# B&R Automation Studio project Kesim (part 4)

#### ManuelAxis.st
```iecst
(*********************************************************************************
 * Copyright:
 * Author:    baranc
 * Created:   October 16, 2025/1:34 PM
 *********************************************************************************)

ACTION ManuelAxis:

	//==================================================
	//		eksenlerin hatalarýnýn sýfýrlanmasý.
	//==================================================
	IF gCommUnit.Main.In.MachineReset THEN
		FOR _i:=0 TO MAX_AX_NR_MIN1 DO
			IF gAxBasic[_i].Error THEN
				gAxBasic[_i].ErrorReset := TRUE;
			END_IF;

		END_FOR
	ELSE
		FOR _i:=0 TO MAX_AX_NR_MIN1 DO
			IF EDGEPOS(gAxBasic[_i].Error = FALSE) THEN //mo25.11.29
				gAxBasic[_i].ErrorReset := FALSE;
			END_IF;
		END_FOR
	END_IF;

	//==================================================
	//		Speed Override
	//==================================================

	gHMI.Diagnosis.SpeedOverride := LREAL_TO_REAL( fbDepthSpeedOverride_0.Out.VelocityOverride) ;

	//==================================================
	//		Aktuel Kenar Hizi
	//==================================================

	IF(gAxBasic[AX_VACUUM].Velocity <> 0 AND gAxBasic[AX_HEAD_Y].Velocity = 0) THEN // movement just in X direction
		gHMI.Diagnosis.ActSealingSpeed := gAxBasic[AX_VACUUM].Velocity;
		IF gAxBasic[AX_VACUUM].Velocity > 1 THEN
	  		gHMI.Widget.MoveHead.Image		:= 'Media/CMS/right.png' ;
		ELSIF gAxBasic[AX_VACUUM].Velocity < -1		THEN

			gHMI.Widget.MoveHead.Image		:= 'Media/CMS/left.png' ;
		END_IF;
	ELSIF (gAxBasic[AX_HEAD_Y].Velocity <> 0 AND gAxBasic[AX_VACUUM].Velocity = 0) THEN // movement just in Y direction
		gHMI.Diagnosis.ActSealingSpeed  := gAxBasic[AX_HEAD_Y].Velocity;
		IF gAxBasic[AX_HEAD_Y].Velocity > 1 THEN
			gHMI.Widget.MoveHead.Image		:= 'Media/CMS/up.png' ;
		ELSIF gAxBasic[AX_HEAD_Y].Velocity < -1		THEN
			gHMI.Widget.MoveHead.Image		:= 'Media/CMS/down.png' ;
		END_IF;
	ELSE	// any other situation - both axes are without motion or moving together - dyn. speed is 0
		gHMI.Diagnosis.ActSealingSpeed  := 0;
		gHMI.Widget.MoveHead.Image		:= 'Media/CMS/none2.png' ;
	END_IF // end of dynamic speed

	//==================================================
	//		Manual hiz ve pos için gerekli degskenlerin atanmasi.
	//==================================================
	IF gPML[0].ModeID = PML_MODE_MAN AND gPML[0].StateCurrent = mpPACKML_STATE_IDLE  THEN

		FOR _i:=0  TO MAX_AX_NR_MIN1 DO
			IF _i >= AX_ENTRY1 AND _i <= AX_EXIT8 THEN //bc25.10.15
				IF (Loc.SelectedStatus.Entrys OR Loc.SelectedStatus.Exits) AND gHMI.Selected.Ax[AX_VACUUM] THEN // Vacuum with conveyors speed

					gAxBasicPar[_i].Velocity 	 		:= gRecData.Manual.Ax[AX_VACUUM].Speed;
					gAxBasicPar[_i].Jog.Velocity 		:= gRecData.Manual.Ax[AX_VACUUM].Speed;
					gAxBasicPar[_i].Jog.Acceleration	:= gRecData.Manual.Ax[AX_VACUUM].Speed * gACCFactor;
					gAxBasicPar[_i].Jog.Deceleration 	:= gRecData.Manual.Ax[AX_VACUUM].Speed * gACCFactor;
					gAxBasicPar[_i].Deceleration 		:= gRecData.Manual.Ax[AX_VACUUM].Speed * gACCFactor;
					gAxBasicPar[_i].Acceleration 		:= gRecData.Manual.Ax[AX_VACUUM].Speed * gACCFactor;
				ELSE
					gAxBasicPar[_i].Velocity 	 		:= gRecData.Manual.Ax[AX_ENTRY1].Speed;
					gAxBasicPar[_i].Jog.Velocity 		:= gRecData.Manual.Ax[AX_ENTRY1].Speed;
					gAxBasicPar[_i].Jog.Acceleration	:= gRecData.Manual.Ax[AX_ENTRY1].Speed * gACCFactor;
					gAxBasicPar[_i].Jog.Deceleration 	:= gRecData.Manual.Ax[AX_ENTRY1].Speed * gACCFactor;
					gAxBasicPar[_i].Deceleration 		:= gRecData.Manual.Ax[AX_ENTRY1].Speed * gACCFactor;
					gAxBasicPar[_i].Acceleration 		:= gRecData.Manual.Ax[AX_ENTRY1].Speed * gACCFactor;
				END_IF;

			ELSIF _i <> AX_HYD THEN
				IF NOT gCommUnit.Main.Status.HYD_MIXER_Y_C_AX AND ( _i = AX_HEAD_C OR _i = AX_HEAD_Y) THEN
					gAxBasicPar[_i].Velocity  			 := gRecData.Manual.Ax[_i].Speed;
					gAxBasicPar[_i].Jog.Velocity 		 := gRecData.Manual.Ax[_i].Speed;
					gAxBasicPar[_i].Jog.Acceleration 	 := gRecData.Manual.Ax[_i].Speed * gACCFactor ;
					gAxBasicPar[_i].Jog.Deceleration 	 := gRecData.Manual.Ax[_i].Speed * gACCFactor ;
					gAxBasicPar[_i].Position    		 := gRecData.Manual.Ax[_i].Pos ;
					gAxBasicPar[_i].Deceleration		 := gRecData.Manual.Ax[_i].Speed * gACCFactor ;
					gAxBasicPar[_i].Acceleration		 := gRecData.Manual.Ax[_i].Speed * gACCFactor ;
				ELSIF ( _i <> AX_HEAD_C OR _i <> AX_HEAD_Y) THEN
					gAxBasicPar[_i].Velocity  			 := gRecData.Manual.Ax[_i].Speed;
					gAxBasicPar[_i].Jog.Velocity 		 := gRecData.Manual.Ax[_i].Speed;
					gAxBasicPar[_i].Jog.Acceleration 	 := gRecData.Manual.Ax[_i].Speed * gACCFactor ;
					gAxBasicPar[_i].Jog.Deceleration 	 := gRecData.Manual.Ax[_i].Speed * gACCFactor ;
					gAxBasicPar[_i].Position    		 := gRecData.Manual.Ax[_i].Pos ;
					gAxBasicPar[_i].Deceleration		 := gRecData.Manual.Ax[_i].Speed * gACCFactor ;
					gAxBasicPar[_i].Acceleration		 := gRecData.Manual.Ax[_i].Speed * gACCFactor ;
				END_IF;

			END_IF;

		END_FOR;
		IF  gPML[0].ModeID = PML_MODE_MAN AND gPML[0].StateCurrent = mpPACKML_STATE_IDLE THEN
			IF gRecData.Manual.Ax[AX_EXIT1_BRIDGE_Y].Pos < gFixData.Ax[AX_EXIT1_BRIDGE_Y].Par.Homing.Position THEN
				gRecData.Manual.Ax[AX_EXIT1_BRIDGE_Y].Pos := LREAL_TO_REAL(gFixData.Ax[AX_EXIT1_BRIDGE_Y].Par.Homing.Position);
			END_IF;
		END_IF;

		fbExitBridgeCtrl_0[AS_BRIDGE_EXIT2].In.Parm.Position.Set 	:= gRecData.Manual.Bridge[AS_BRIDGE_EXIT2].Pos;
		fbExitBridgeCtrl_0[AS_BRIDGE_EXIT2].In.Parm.Speed.SpeedMan 	:= gRecData.Manual.Ax[AX_EXIT1_BRIDGE_Y].Speed * 0.25; // servo eksenin max hizi ile asenktron eksenin max hizi arasindaki oran

		fbExitBridgeCtrl_0[AS_BRIDGE_EXIT3].In.Parm.Position.Set 	:= gRecData.Manual.Bridge[AS_BRIDGE_EXIT3].Pos;
		fbExitBridgeCtrl_0[AS_BRIDGE_EXIT3].In.Parm.Speed.SpeedMan 	:= gRecData.Manual.Ax[AX_EXIT1_BRIDGE_Y].Speed * 0.25;

		fbExitBridgeCtrl_0[AS_BRIDGE_EXIT4].In.Parm.Position.Set 	:= gRecData.Manual.Bridge[AS_BRIDGE_EXIT4].Pos;
		fbExitBridgeCtrl_0[AS_BRIDGE_EXIT4].In.Parm.Speed.SpeedMan 	:= gRecData.Manual.Ax[AX_EXIT1_BRIDGE_Y].Speed * 0.25;

	END_IF

	//==================================================
	//		Y EKSEN GUVENLI POZISYONDA DEGIL. EXIT 1 IN YADA ENTRY 1 OUT SENSORU GORURSE VAKUM VE KONVEYOR HIZLARI DÜSSSÜN.
	//==================================================
	IF gAxBasic[AX_HEAD_Y].Position >10 AND gPML[0].ModeID = PML_MODE_MAN THEN
		IF gIO.In.Entry[ENTR1_UNIT].OutSens OR gIO.In.Exit[EXIT1_UNIT].Conv.InSens THEN
			IF gHMI.Selected.Ax[AX_VACUUM] AND gIO.In.Sealing.X2VacuumOK THEN
				gRecData.Manual.Ax[AX_VACUUM].Speed		:= 50 ;
				IF gAxBasic[AX_VACUUM].MoveActive AND gAxBasicPar[AX_VACUUM].Velocity <> gRecData.Manual.Ax[AX_VACUUM].Speed THEN

					gAxBasicPar[AX_VACUUM].Velocity 	 		:= gRecData.Manual.Ax[AX_VACUUM].Speed;
					gAxBasicPar[AX_VACUUM].Jog.Velocity 		:= gRecData.Manual.Ax[AX_VACUUM].Speed;
					gAxBasicPar[AX_VACUUM].Jog.Acceleration		:= gRecData.Manual.Ax[AX_VACUUM].Speed * 5;
					gAxBasicPar[AX_VACUUM].Jog.Deceleration 	:= gRecData.Manual.Ax[AX_VACUUM].Speed * 5;
					gAxBasicPar[AX_VACUUM].Deceleration 		:= gRecData.Manual.Ax[AX_VACUUM].Speed * 5;
					gAxBasicPar[AX_VACUUM].Acceleration 		:= gRecData.Manual.Ax[AX_VACUUM].Speed * 5;

					gAxBasicPar[AX_ENTRY1].Velocity 	 		:= gRecData.Manual.Ax[AX_VACUUM].Speed;
					gAxBasicPar[AX_ENTRY1].Jog.Velocity 		:= gRecData.Manual.Ax[AX_VACUUM].Speed;
					gAxBasicPar[AX_ENTRY1].Jog.Acceleration		:= gRecData.Manual.Ax[AX_VACUUM].Speed * 5;
					gAxBasicPar[AX_ENTRY1].Jog.Deceleration 	:= gRecData.Manual.Ax[AX_VACUUM].Speed * 5;
					gAxBasicPar[AX_ENTRY1].Deceleration 		:= gRecData.Manual.Ax[AX_VACUUM].Speed * 5;
					gAxBasicPar[AX_ENTRY1].Acceleration 		:= gRecData.Manual.Ax[AX_VACUUM].Speed * 5;

					gAxBasicPar[AX_EXIT1].Velocity 	 			:= gRecData.Manual.Ax[AX_VACUUM].Speed;
					gAxBasicPar[AX_EXIT1].Jog.Velocity 			:= gRecData.Manual.Ax[AX_VACUUM].Speed;
					gAxBasicPar[AX_EXIT1].Jog.Acceleration		:= gRecData.Manual.Ax[AX_VACUUM].Speed * 5;
					gAxBasicPar[AX_EXIT1].Jog.Deceleration 		:= gRecData.Manual.Ax[AX_VACUUM].Speed * 5;
					gAxBasicPar[AX_EXIT1].Deceleration 			:= gRecData.Manual.Ax[AX_VACUUM].Speed * 5;
					gAxBasicPar[AX_EXIT1].Acceleration 			:= gRecData.Manual.Ax[AX_VACUUM].Speed * 5;

					IF (gAxBasic[AX_VACUUM].MoveActive AND gAxBasicPar[AX_VACUUM].Velocity <> gAxBasic[AX_VACUUM].Velocity)  THEN
						gAxBasic[AX_VACUUM].Update 	:= TRUE ;
					END_IF;

					IF (gAxBasic[AX_ENTRY1].MoveActive AND gAxBasicPar[AX_ENTRY1].Velocity <> gAxBasic[AX_ENTRY1].Velocity)  THEN
						gAxBasic[AX_ENTRY1].Update 	:= TRUE ;
					END_IF;

					IF (gAxBasic[AX_EXIT1].MoveActive AND gAxBasicPar[AX_EXIT1].Velocity <> gAxBasic[AX_EXIT1].Velocity) THEN
						gAxBasic[AX_EXIT1].Update	:= TRUE ;
					END_IF;
				END_IF
				IF gAxBasic[AX_VACUUM].UpdateDone THEN
					gAxBasic[AX_VACUUM].Update 	:= FALSE ;
				END_IF;
				IF gAxBasic[AX_ENTRY1].UpdateDone THEN
					gAxBasic[AX_ENTRY1].Update 	:= FALSE ;
				END_IF;
				IF gAxBasic[AX_EXIT1].UpdateDone THEN
					gAxBasic[AX_EXIT1].Update	:= FALSE ;
				END_IF;

			ELSIF gHMI.Selected.Ax[AX_ENTRY1] OR gHMI.Selected.Ax[AX_EXIT1] THEN
				gRecData.Manual.Ax[AX_ENTRY1].Speed		:= 50 ;

				gAxBasicPar[AX_ENTRY1].Velocity 	 		:= gRecData.Manual.Ax[AX_ENTRY1].Speed;
				gAxBasicPar[AX_ENTRY1].Jog.Velocity 		:= gRecData.Manual.Ax[AX_ENTRY1].Speed;
				gAxBasicPar[AX_ENTRY1].Jog.Acceleration		:= gRecData.Manual.Ax[AX_ENTRY1].Speed * 5;
				gAxBasicPar[AX_ENTRY1].Jog.Deceleration 	:= gRecData.Manual.Ax[AX_ENTRY1].Speed * 5;
				gAxBasicPar[AX_ENTRY1].Deceleration 		:= gRecData.Manual.Ax[AX_ENTRY1].Speed * 5;
				gAxBasicPar[AX_ENTRY1].Acceleration 		:= gRecData.Manual.Ax[AX_ENTRY1].Speed * 5;

				gAxBasicPar[AX_EXIT1].Velocity 	 			:= gRecData.Manual.Ax[AX_ENTRY1].Speed;
				gAxBasicPar[AX_EXIT1].Jog.Velocity 			:= gRecData.Manual.Ax[AX_ENTRY1].Speed;
				gAxBasicPar[AX_EXIT1].Jog.Acceleration		:= gRecData.Manual.Ax[AX_ENTRY1].Speed * 5;
				gAxBasicPar[AX_EXIT1].Jog.Deceleration 		:= gRecData.Manual.Ax[AX_ENTRY1].Speed * 5;
				gAxBasicPar[AX_EXIT1].Deceleration 			:= gRecData.Manual.Ax[AX_ENTRY1].Speed * 5;
				gAxBasicPar[AX_EXIT1].Acceleration 			:= gRecData.Manual.Ax[AX_ENTRY1].Speed * 5;

				IF (gAxBasic[AX_ENTRY1].MoveActive AND gAxBasicPar[AX_ENTRY1].Velocity <> gAxBasic[AX_ENTRY1].Velocity)  THEN
					gAxBasic[AX_ENTRY1].Update 	:= TRUE ;
				END_IF;

				IF (gAxBasic[AX_EXIT1].MoveActive AND gAxBasicPar[AX_EXIT1].Velocity <> gAxBasic[AX_EXIT1].Velocity) THEN
					gAxBasic[AX_EXIT1].Update	:= TRUE ;
				END_IF;
				IF gAxBasic[AX_ENTRY1].UpdateDone THEN
					gAxBasic[AX_ENTRY1].Update 	:= FALSE ;
				END_IF;
				IF gAxBasic[AX_EXIT1].UpdateDone THEN
					gAxBasic[AX_EXIT1].Update	:= FALSE ;
				END_IF;
			END_IF;

		END_IF;
	END_IF;
	//	gAxBasicPar[AX_EXIT1]();
	//	gAxBasic[AX_EXIT1]();

	//==================================================
	//		EXIT CONV SEÇILI MI ?
	//==================================================
	Loc.SelectedStatus.Exits := FALSE;
	FOR _i := AX_EXIT1 TO AX_EXIT8 DO

		IF gHMI.Selected.Ax[_i] THEN
			Loc.SelectedStatus.Exits := TRUE;
		END_IF;

	END_FOR;

	//==================================================
	//		ENTRY CONV SEÇILI MI ?
	//==================================================
	Loc.SelectedStatus.Entrys := FALSE;
	FOR _i:=AX_ENTRY1 TO AX_ENTRY4 DO

		IF gHMI.Selected.Ax[_i] THEN
			Loc.SelectedStatus.Entrys := TRUE;
		END_IF;

	END_FOR;

	//==================================================
	//	    AS KOPRULER SEÇILI MI ?
	//==================================================
	Loc.SelectedStatus.Bridges := FALSE;
	FOR _i:=AS_BRIDGE_EXIT2 TO AS_BRIDGE_EXIT8 DO

		IF gHMI.Selected.Bridge[_i] THEN
			Loc.SelectedStatus.Bridges := TRUE;
		END_IF;
	END_FOR;

	//==================================================
	//	     Konveyor Giris Z Eksenleri SEÇILI MI ?
	//==================================================
	Loc.SelectedStatus.EntryThicness := FALSE;
	FOR _i:=ENTR1_UNIT TO ENTR4_UNIT DO

		IF gHMI.Selected.Thick.Entry[_i] THEN
			Loc.SelectedStatus.EntryThicness := TRUE;
		END_IF;
	END_FOR;

	//==================================================
	//	     Konveyor Çikis Z Eksenleri SEÇILI MI ?
	//==================================================
	Loc.SelectedStatus.ExitThicness := FALSE;
	FOR _i:=EXIT1_UNIT TO EXIT8_UNIT DO

		IF gHMI.Selected.Thick.Exit[_i] THEN
			Loc.SelectedStatus.ExitThicness := TRUE;
		END_IF;
	END_FOR;

	//==================================================
	//		C EKSEN SEÇILEMEZ
	//==================================================
	gHMI.Diagnosis.Ax[AX_HEAD_C].Block :=

	NOT gAxBasic[AX_HEAD_C].PowerOn OR
	NOT(Loc.SelectedStatus.Entrys OR
	Loc.SelectedStatus.Exits OR
	Loc.SelectedStatus.Bridges OR
	gHMI.Selected.Ax[AX_EXIT1_BRIDGE_Y	] OR
	gHMI.Selected.Ax[AX_HEAD_Z] OR
	gHMI.Selected.Ax[AX_VACUUM] OR
	gHMI.Selected.Ax[AX_HEAD_Y] OR
	gPML[0].ModeID = PML_MODE_AUTO OR
	Loc.SelectedStatus.ExitThicness ) ;

	//==================================================
	//		Y EKSEN SEÇILEMEZ
	//==================================================
	gHMI.Diagnosis.Ax[AX_HEAD_Y].Block :=
	NOT gAxBasic[AX_HEAD_Y].PowerOn OR
	NOT (Loc.SelectedStatus.Entrys OR
	Loc.SelectedStatus.Exits OR
	Loc.SelectedStatus.Bridges OR
	gHMI.Selected.Ax[AX_EXIT1_BRIDGE_Y	] OR
	gHMI.Selected.Ax[AX_HEAD_Z] OR
	gHMI.Selected.Ax[AX_VACUUM] OR
	gHMI.Selected.Ax[AX_HEAD_C] OR
	gPML[0].ModeID = PML_MODE_AUTO OR
	Loc.SelectedStatus.ExitThicness ) ;

	//==================================================
	//		Z EKSEN SEÇILEMEZ
	//==================================================
	gHMI.Diagnosis.Ax[AX_HEAD_Z].Block :=
	NOT gAxBasic[AX_HEAD_Z].PowerOn OR
	NOT (Loc.SelectedStatus.Entrys OR
	Loc.SelectedStatus.Exits OR
	Loc.SelectedStatus.Bridges OR
	gHMI.Selected.Ax[AX_EXIT1_BRIDGE_Y	] OR
	gHMI.Selected.Ax[AX_HEAD_Y] OR
	gHMI.Selected.Ax[AX_VACUUM] OR
	gHMI.Selected.Ax[AX_HEAD_C] OR
	gPML[0].ModeID = PML_MODE_AUTO OR
	Loc.SelectedStatus.ExitThicness ) ;

	//==================================================
	//		VAKUM EKSENI SEÇILEMEZ
	//==================================================
	gHMI.Diagnosis.Ax[AX_VACUUM].Block :=
	NOT gAxBasic[AX_VACUUM].PowerOn OR
	NOT (Loc.SelectedStatus.Bridges OR
	gHMI.Selected.Ax[AX_EXIT1_BRIDGE_Y	] OR
	gHMI.Selected.Ax[AX_HEAD_Y] OR
	gHMI.Selected.Ax[AX_HEAD_Z] OR
	gHMI.Selected.Ax[AX_HEAD_C] OR
	gPML[0].ModeID = PML_MODE_AUTO OR
	Loc.SelectedStatus.ExitThicness );

	//==================================================
	//		KOPRU 1(Servo Eksen) SEÇILEMEZ
	//==================================================
	gHMI.Diagnosis.Ax[AX_EXIT1_BRIDGE_Y].Block :=
	NOT gAxBasic[AX_EXIT1_BRIDGE_Y].PowerOn OR
	NOT( Loc.SelectedStatus.Entrys OR
	Loc.SelectedStatus.Exits OR
	gHMI.Selected.Ax[AX_VACUUM	] OR
	gHMI.Selected.Ax[AX_HEAD_Y] OR
	gHMI.Selected.Ax[AX_HEAD_Z] OR
	gHMI.Selected.Ax[AX_HEAD_C] OR
	gPML[0].ModeID = PML_MODE_AUTO OR
	Loc.SelectedStatus.ExitThicness ) ;

	//==================================================
	//		CONV SEÇILEMEZ
	//==================================================
	gHMI.Diagnosis.Ax[AX_ENTRY1].Block :=

	NOT (Loc.SelectedStatus.Bridges OR
	gHMI.Selected.Ax[AX_EXIT1_BRIDGE_Y	] OR
	gHMI.Selected.Ax[AX_HEAD_Y] OR
	gHMI.Selected.Ax[AX_HEAD_Z] OR
	gHMI.Selected.Ax[AX_HEAD_C] OR
	gPML[0].ModeID = PML_MODE_AUTO OR
	Loc.SelectedStatus.ExitThicness ) ;

	//==================================================
	//		KOPRULER(AS) SEÇILEMEZ
	//======================W============================
	gHMI.Diagnosis.Brdige[AS_BRIDGE_EXIT2].Block :=
	gPML[0].ModeID = PML_MODE_AUTO OR
	NOT( Loc.SelectedStatus.Entrys OR
	Loc.SelectedStatus.Exits OR
	gHMI.Selected.Ax[AX_VACUUM	] OR
	gHMI.Selected.Ax[AX_HEAD_Y] OR
	gHMI.Selected.Ax[AX_HEAD_Z] OR
	gHMI.Selected.Ax[AX_HEAD_C] OR
	gPML[0].ModeID = PML_MODE_AUTO OR
	Loc.SelectedStatus.ExitThicness ) ;

	//==================================================
	//		KALINLIK(AS) SEÇILEMEZ
	//======================W============================
	gHMI.Diagnosis.EntryThickness[ENTR1_UNIT].Block :=
	gPML[0].ModeID = PML_MODE_AUTO OR
	NOT( Loc.SelectedStatus.Entrys OR
	Loc.SelectedStatus.Exits OR
	gHMI.Selected.Ax[AX_VACUUM	] OR
	gHMI.Selected.Ax[AX_HEAD_Y] OR
	gHMI.Selected.Ax[AX_HEAD_Z] OR
	gHMI.Selected.Ax[AX_HEAD_C] OR
	gPML[0].ModeID = PML_MODE_AUTO OR
	Loc.SelectedStatus.Bridges ) ;

	//==================================================
	//		Vakum Seçili Degil. Vakum Sinyali var. Xler hareket etmesin.
	//==================================================

	Loc.SelectedStatus.VacuumWithConv := TRUE;

	IF gHMI.Selected.Conv.Entry[ENTR1_UNIT] AND NOT gHMI.Selected.Ax[AX_VACUUM] AND gIO.In.Sealing.X2VacuumOK THEN
		Loc.SelectedStatus.VacuumWithConv := FALSE;
	END_IF;

	IF gHMI.Selected.Conv.Entry[ENTR2_UNIT] AND NOT gHMI.Selected.Ax[AX_VACUUM] AND gIO.In.Sealing.X2VacuumOK AND gIO.In.Entry[ENTR2_UNIT].OutSens THEN
		Loc.SelectedStatus.VacuumWithConv := FALSE;
	END_IF;

	IF gHMI.Selected.Conv.Entry[EXIT1_UNIT] AND NOT gHMI.Selected.Ax[AX_VACUUM] AND gIO.In.Sealing.X2VacuumOK THEN
		Loc.SelectedStatus.VacuumWithConv := FALSE;
	END_IF;

	IF gHMI.Selected.Conv.Entry[EXIT2_UNIT] AND NOT gHMI.Selected.Ax[AX_VACUUM] AND gIO.In.Sealing.X2VacuumOK AND gIO.In.Exit[EXIT2_UNIT].Conv.InSens THEN
		Loc.SelectedStatus.VacuumWithConv := FALSE;
	END_IF;

	//	IF Loc.SelectedStatus.VacuumWithConv = FALSE AND (gHMI.Cmd.Jog.Neg OR gHMI.Cmd.Jog.Pos)  THEN
	//		gCommUnit.EntryMain.Out.ConvNotMoved      := TRUE;
	//		gAlert.Info.IDX[INFO_VACUUM_NOT_SELECTED] := TRUE;
	//	ELSE
	//		gCommUnit.EntryMain.Out.ConvNotMoved      := FALSE;
	//	END_IF;

	//==================================================
	//		Vakum var.Vakum Ekseni seçili. Kovveyorler seçili olmadan hareket verilmesin.
	//==================================================
	//	Loc.SelectedStatus.ConvWithVacuum				:= TRUE;

	IF gIO.In.Sealing.X2VacuumOK AND EDGEPOS(gHMI.Selected.Ax[AX_ENTRY1] OR gHMI.Selected.Ax[AX_EXIT1] OR gHMI.Selected.Ax[AX_VACUUM]) THEN
		gHMI.Selected.Ax[AX_ENTRY1]	:= TRUE;
		gHMI.Selected.Ax[AX_EXIT1]	:= TRUE;
		gHMI.Selected.Ax[AX_VACUUM]	:= TRUE;
	END_IF;

	//	IF gHMI.Selected.Ax[AX_VACUUM] AND NOT gHMI.Selected.Ax[AX_ENTRY2] AND gIO.In.Sealing.X2VacuumOK AND gIO.In.Entry[ENTR2_UNIT].OutSens THEN
	//	  	Loc.SelectedStatus.ConvWithVacuum				:= FALSE;
	//	END_IF;
	//
	//	IF gHMI.Selected.Ax[AX_VACUUM] AND NOT gHMI.Selected.Ax[AX_ENTRY1] AND gIO.In.Sealing.X2VacuumOK THEN
	//		Loc.SelectedStatus.ConvWithVacuum				:= FALSE;
	//	END_IF;
	//
	//	IF gHMI.Selected.Ax[AX_VACUUM] AND NOT gHMI.Selected.Ax[AX_EXIT1] AND gIO.In.Sealing.X2VacuumOK THEN
	//		Loc.SelectedStatus.ConvWithVacuum				:= FALSE;
	//	END_IF;
	//
	//	IF gHMI.Selected.Ax[AX_VACUUM] AND NOT gHMI.Selected.Ax[AX_EXIT2] AND gIO.In.Sealing.X2VacuumOK AND gIO.In.Exit[EXIT2_UNIT].Conv.InSens THEN
	//		Loc.SelectedStatus.ConvWithVacuum				:= FALSE;
	//	END_IF;

	//	IF Loc.SelectedStatus.ConvWithVacuum  = FALSE THEN
	//		gCommUnit.EntryMain.Out.VacuumNotMoved      := TRUE;
	//		gAlert.Info.IDX[INFO_CONV_NOT_SELECTED] 	:= TRUE;
	//	ELSE
	//		gCommUnit.EntryMain.Out.VacuumNotMoved      := FALSE;
	//	END_IF

	//==================================================
	//		Vakumlu iken vakum ekseni - limite geldiyse konveyor hareket olmasin..
	//==================================================

	//==================================================
	//		RESETE BASILINCA TÜM SEÇIMLERI KALDIRSIN
	//==================================================

	TON_ResetAxis.IN	:= gCommUnit.Main.In.MachineReset;
	TON_ResetAxis.PT	:= T#0.3S;
	TON_ResetAxis();

	IF TON_ResetAxis.Q OR EDGEPOS(gPML[0].ModeID = PML_MODE_AUTO) THEN

		FOR _i := 0 TO MAX_AX_NR_MIN1 DO
			gHMI.Selected.Ax[_i ] := FALSE;
		END_FOR;

		FOR _i := AS_BRIDGE_EXIT2 TO AS_BRIDGE_EXIT8 DO
			gHMI.Selected.Bridge[_i ] := FALSE;
		END_FOR;

		FOR _i := EXIT1_UNIT TO EXIT8_UNIT DO
			gHMI.Selected.Thick.Exit[_i ] := FALSE;
		END_FOR;

		FOR _i := ENTR1_UNIT TO ENTR4_UNIT DO
			gHMI.Selected.Thick.Entry[_i ] := FALSE;
		END_FOR;

	END_IF

END_ACTION
```

#### MaxMinValue.st
```iecst
(*********************************************************************************
 * Copyright:
 * Author:    baranc
 * Created:   October 20, 2025/9:22 AM
 *********************************************************************************)

ACTION MaxMinValue:
	//==================================================
	//		Cam boyutu max deđerleri
	//==================================================
	gHMI.Widget.GlassXSize.Max := gFixData.HwConfig.EntryUnitInstalled* gFixData.HwConfig.ConvLength;
	gHMI.Widget.GlassXSize.Max := gFixData.HwConfig.EntryUnitInstalled* gFixData.HwConfig.ConvLength;
	gHMI.Widget.Pressure.Min   := gFixData.Material[gFixData.Config.Material].AFilling[gHydr.In.ActiveUnit-1] + 20 ;
	gHMI.Widget.ProductionDaily.Max	:= MAX(gFixData.Production.Daily.DoubleGlass,gFixData.Production.Daily.TripleGlass) + 50 ;
	gHMI.Widget.ProductionMonth.Max	:= MAX(gFixData.Production.Month.DoubleGlass,gFixData.Production.Month.TripleGlass) + 50 ;
	gHMI.Widget.ProductionTotal.Max	:= MAX(gFixData.Production.Total.DoubleGlass,gFixData.Production.Total.TripleGlass) + 50 ;

END_ACTION
```

#### ManualDevice.st
```iecst
(*********************************************************************************
 * Copyright:
 * Author:    baranc
 * Created:   November 3, 2025/4:10 PM
 *********************************************************************************)

ACTION ManualDevice:

	IF fbVacuumCtrl_0.In.Cmd.VacuumOn = TRUE  AND  fbVacuumCtrl_0.Out.CommandDone THEN
		fbVacuumCtrl_0.In.Cmd.VacuumOn := FALSE;
	END_IF;
	IF gHMI.Cmd.Manual.VacuumGlass THEN
		fbVacuumCtrl_0.In.Cmd.VacuumOn := TRUE;
		(*fbVacuumCtrl_0.In.Cmd.VacuumOff := FALSE;*)
	END_IF;

	IF fbVacuumCtrl_0.In.Cmd.VacuumOff = TRUE  AND  fbVacuumCtrl_0.Out.CommandDone = TRUE THEN
		gHMI.Selected.Ax[AX_VACUUM] 	:= FALSE;
		fbVacuumCtrl_0.In.Cmd.VacuumOff := FALSE;
	END_IF;
	IF gHMI.Cmd.Manual.ReleaseGlass THEN
		(*fbVacuumCtrl_0.In.Cmd.VacuumOn := FALSE;*)
		fbVacuumCtrl_0.In.Cmd.VacuumOff := TRUE;
	END_IF;

	fbVacuumCtrl_0();

	FOR _k := 0 TO Max_Manual_Device DO
		fbManualDeviceCtrl[_k].In.bEnable := TRUE;
		fbManualDeviceCtrl[_k].In.bResettable := TRUE ;
		fbManualDeviceCtrl[_k].In.bEmergencyStop := TRUE;
		fbManualDeviceCtrl[_k].In.bManualMode := gPML[0].ModeID = PML_MODE_MAN;
	END_FOR;

	//==================================================
	//		Manual Device örnek kullaným.
	//==================================================
	//	fbManualDeviceCtrl[UNIT_LargeSpatulaPiston].In.bInput := Sinyali tetikleyecek deđiţken buraya yazýlýr;
	//	fbManualDeviceCtrl[UNIT_LargeSpatulaPiston].In.bSensor := Sensore bađlý ;
	//	Kontrol edilecek çýkýţ. := fbManualDeviceCtrl[UNIT_LargeSpatulaPiston].Out.bOutput ;
	//  fbManualDeviceCtrl[UNIT_LargeSpatulaPiston]();

	//==================================================
	//		Large Spatula Piston Manual
	//==================================================
	//	fbManualDeviceCtrl[UNIT_LargeSpatulaPiston].In.bInput := gHMI.Cmd.Manual.LargeSpatulaPiston;
	//	fbManualDeviceCtrl[UNIT_LargeSpatulaPiston].In.bSensor := FALSE; (*gIO.In.Sealing.SpatulaBigPistonBack*) ;
	//	gIO.Out.Sealing.SpatulaBigPistonFrw := fbManualDeviceCtrl[UNIT_LargeSpatulaPiston].Out.bOutput ;
	//	fbManualDeviceCtrl[UNIT_LargeSpatulaPiston]();

	IF EDGEPOS(gHMI.Cmd.Manual.LargeSpatulaPiston) THEN
		fbScrapperProcess_0.In.Cmd.Start:= TRUE;
	END_IF
	IF EDGEPOS(NOT gHMI.Cmd.Manual.LargeSpatulaPiston) THEN
		fbScrapperProcess_0.In.Cmd.Start:= FALSE;
	END_IF;

	//==================================================
	//		Small Spatula Piston Manual
	//==================================================
	//	fbManualDeviceCtrl[UNIT_SmallSpatulaPiston].In.bInput := gHMI.Cmd.Manual.SmallSpatulaPiston;
	//	fbManualDeviceCtrl[UNIT_SmallSpatulaPiston].In.bSensor := FALSE; (*gIO.In.Sealing.SpatulaSmallPistonBack*) ;
	//	gIO.Out.Sealing.SpatulaSmallPistonFrw := fbManualDeviceCtrl[UNIT_SmallSpatulaPiston].Out.bOutput ;
	//	fbManualDeviceCtrl[UNIT_SmallSpatulaPiston]();
	IF EDGEPOS(NOT gHMI.Cmd.Manual.SmallSpatulaPiston) THEN
		fbScrapperProcess_0.In.Cmd.EdgeLast:= FALSE;
		fbScrapperProcess_0.In.Cmd.Start:= FALSE;

	END_IF;
	IF EDGEPOS(gHMI.Cmd.Manual.SmallSpatulaPiston) THEN
		fbScrapperProcess_0.In.Cmd.EdgeLast:= TRUE;
		fbScrapperProcess_0.In.Cmd.Start:= TRUE;

	END_IF;

	//==================================================
	//		DepthForward
	//==================================================
	fbManualDeviceCtrl[UNIT_DepthValve].In.bInput := gHMI.Cmd.Manual.DepthForward;
	fbManualDeviceCtrl[UNIT_DepthValve].In.bSensor := FALSE ;
	gIO.Out.Sealing.DepthForward := fbManualDeviceCtrl[UNIT_DepthValve].Out.bOutput ;
	fbManualDeviceCtrl[UNIT_DepthValve]();

	//==================================================
	//		Material Out Valve
	//==================================================
	fbManualDeviceCtrl[UNIT_MaterialOutValve].In.bInput := gHMI.Cmd.Manual.MaterialOutValve;
	fbManualDeviceCtrl[UNIT_MaterialOutValve].In.bSensor := FALSE ;
	gIO.Out.Hydr.General.MaterialOpenValve := fbManualDeviceCtrl[UNIT_MaterialOutValve].Out.bOutput ;
	fbManualDeviceCtrl[UNIT_MaterialOutValve]();

END_ACTION
```

#### Home.st
```iecst
(*********************************************************************************
 * Copyright:
 * Author:    baranc
 * Created:   October 27, 2025/7:52 AM
 *********************************************************************************)

ACTION Home:

	//========================================================================================
	// AX_HEAD_C Servo Axis  Home Offset ini Hesaplama
	//========================================================================================
	CASE StateAbsCHomeOffset OF
		0: //WAIT_ABS_HOME_CMD
			IF gHMI.Cmd.bHome.Ax[AX_HEAD_C] AND NOT gAxBasic[ AX_HEAD_C].Error THEN
				gAxBasic[ AX_HEAD_C].Home 		:= FALSE;
				StateAbsCHomeOffset := 10;
			ELSE
				gHMI.Cmd.bHome.Ax[AX_HEAD_C] := FALSE;
			END_IF

		10: // POWER_ON_CHK
			IF (gAxBasic[ AX_HEAD_C].PowerOn = FALSE) THEN
				gAxBasic[ AX_HEAD_C].Power := TRUE;
			ELSIF gAxBasic[ AX_HEAD_C].PowerOn THEN
				StateAbsCHomeOffset := 20;
			END_IF

		20:// DIRECT HOME
			// Once Eksen Homelanir
			gAxBasicPar[AX_HEAD_C].Homing.Mode 		:= mcHOMING_DIRECT;
			gAxBasicPar[ AX_HEAD_C].Homing.Position	:= 0;
			IF gFixData.Ax[ AX_HEAD_C].Enabled AND NOT gAxBasic[ AX_HEAD_C].CommandBusy THEN
				gAxBasic[ AX_HEAD_C].Home := TRUE;
				StateAbsCHomeOffset := 25;
			END_IF;

		25: (* Wait Home *)
			IF (gAxBasic[ AX_HEAD_C].IsHomed) THEN
				gAxBasic[ AX_HEAD_C].Home 		:= FALSE;
				gFixData.MultiturnEncOffsets.AX_C_EncOffset := ( gAxBasic[ AX_HEAD_C].Position );
				StateAbsCHomeOffset := 30;
			END_IF

		30: // MC_ReadParameter
			// Ham Enkoder Degeri Okunur
			MC_ReadParameterC_FB.Axis 			:= ADR(gAxis_HeadC);
			MC_ReadParameterC_FB.ParameterNumber := mcPAR_HOMING_OFFSET;
			MC_ReadParameterC_FB.Enable 			:= TRUE;
			MC_ReadParameterC_FB();

			// Ham Degere HMI dan Set edilen istenen degere offsetlenir
			IF MC_ReadParameterC_FB.Valid THEN
				MC_ReadParameterC_FB.Enable := FALSE;
				gFixData.MultiturnEncOffsets.AX_C_EncOffset := ( MC_ReadParameterC_FB.Value ) + gFixData.Ax[AX_HEAD_C].Par.Homing.Position;(* HMI Set Deger*)
				StateAbsCHomeOffset 		:= 40;
			END_IF

		40: // mcHOMING_ABSOLUTE
			// Absolute Home Position degeri olarak Homing yapilir
			gAxBasicPar[AX_HEAD_C].Homing.Mode 		:= mcHOMING_ABSOLUTE;
			gAxBasicPar[ AX_HEAD_C].Homing.Position	:= gFixData.MultiturnEncOffsets.AX_C_EncOffset;
			IF gFixData.Ax[ AX_HEAD_C].Enabled AND NOT gAxBasic[ AX_HEAD_C].CommandBusy THEN
				gAxBasic[ AX_HEAD_C].Home := TRUE;
				StateAbsCHomeOffset := 45;
			END_IF;

		45: (* Wait Home *)
			IF (gAxBasic[ AX_HEAD_C].IsHomed) THEN
				gAxBasic[ AX_HEAD_C].Home 		:= FALSE;
				gHMI.Cmd.bHome.Ax[AX_HEAD_C] := FALSE;
				gAxBasic[ AX_HEAD_C].Home  := FALSE;
				StateAbsCHomeOffset 			:= 0;
			END_IF

	END_CASE;

	MC_ReadParameterC_FB();

	//========================================================================================
	// AX_HEAD_Z Servo Axis  Home Offset ini Hesaplama
	//========================================================================================

	CASE StateAbsZHomeOffset OF
		0: //WAIT_ABS_HOME_CMD
			IF gHMI.Cmd.bHome.Ax[AX_HEAD_Z] AND NOT gAxBasic[ AX_HEAD_Z].Error THEN
				gAxBasic[ AX_HEAD_Z].Home 		:= FALSE;
				StateAbsZHomeOffset := 10;
			ELSE
				gHMI.Cmd.bHome.Ax[AX_HEAD_Z] := FALSE;
			END_IF

		10: // POWER_ON_CHK
			IF (gAxBasic[ AX_HEAD_Z].PowerOn = FALSE) THEN
				gAxBasic[ AX_HEAD_Z].Power := TRUE;
			ELSIF gAxBasic[ AX_HEAD_Z].PowerOn THEN
				StateAbsZHomeOffset := 20;
			END_IF

		20:// DIRECT HOME
			// Once Eksen Homelanir
			gAxBasicPar[AX_HEAD_Z].Homing.Mode 		:= mcHOMING_DIRECT;
			gAxBasicPar[ AX_HEAD_Z].Homing.Position	:= 0;
			IF gFixData.Ax[ AX_HEAD_Z].Enabled AND NOT gAxBasic[ AX_HEAD_Z].CommandBusy THEN
				gAxBasic[ AX_HEAD_Z].Home := TRUE;
				StateAbsZHomeOffset := 25;
			END_IF;

		25: (* Wait Home *)
			IF (gAxBasic[ AX_HEAD_Z].IsHomed) THEN
				gAxBasic[ AX_HEAD_Z].Home 		:= FALSE;
				gFixData.MultiturnEncOffsets.AX_Z_EncOffset := ( gAxBasic[ AX_HEAD_Z].Position );
				StateAbsZHomeOffset := 30;
			END_IF

		30: // MC_ReadParameter
			// Ham Enkoder Degeri Okunur
			MC_ReadParameterZ_FB.Axis 			:= ADR(gAxis_HeadZ);
			MC_ReadParameterZ_FB.ParameterNumber := mcPAR_HOMING_OFFSET;
			MC_ReadParameterZ_FB.Enable 			:= TRUE;
			MC_ReadParameterZ_FB();

			// Ham Degere HMI dan Set edilen istenen degere offsetlenir
			IF MC_ReadParameterZ_FB.Valid THEN
				MC_ReadParameterZ_FB.Enable := FALSE;
				gFixData.MultiturnEncOffsets.AX_Z_EncOffset := ( MC_ReadParameterZ_FB.Value ) + gFixData.Ax[AX_HEAD_Z].Par.Homing.Position;(* HMI Set Deger*)
				StateAbsZHomeOffset 		:= 40;
			END_IF

		40: // mcHOMING_ABSOLUTE
			// Absolute Home Position degeri olarak Homing yapilir
			gAxBasicPar[AX_HEAD_Z].Homing.Mode 		:= mcHOMING_ABSOLUTE;
			gAxBasicPar[ AX_HEAD_Z].Homing.Position	:= gFixData.MultiturnEncOffsets.AX_Z_EncOffset;
			IF gFixData.Ax[ AX_HEAD_Z].Enabled AND NOT gAxBasic[ AX_HEAD_Z].CommandBusy THEN
				gAxBasic[ AX_HEAD_Z].Home := TRUE;
				StateAbsZHomeOffset := 45;
			END_IF;

		45: (* Wait Home *)
			IF (gAxBasic[ AX_HEAD_Z].IsHomed) THEN
				gAxBasic[ AX_HEAD_Z].Home 		:= FALSE;
				gHMI.Cmd.bHome.Ax[AX_HEAD_Z] := FALSE;
				gAxBasic[ AX_HEAD_Z].Home  := FALSE;
				StateAbsZHomeOffset 			:= 0;
			END_IF

	END_CASE;

	MC_ReadParameterZ_FB();

	//	//Execture manual
	//	gAxBasicPar[12].Homing.Mode	    := mcHOMING_ABSOLUTE;
	//	gAxBasicPar[12].Homing.Position := gParDataEksen12.Offset;
	//
	//	// power ver
	//	// direct home ver
	//	// mc_readparam cagir.
	//	// gParDataEksen12.Offset  0 olamaz
	//	//motor sökülmedigi sürece çalistirmaya gerek yok
	//	IF MakineAyarlandiHomePozisyonBurasi THEN
	//		MC_ReadParameter_FB.Axis := ADR(gAxis_HeadZ);
	//		MC_ReadParameter_FB.ParameterNumber := mcPAR_HOMING_OFFSET;
	//		MC_ReadParameter_FB.Enable := TRUE;
	//		MC_ReadParameter_FB();
	//	END_IF;
	//	IF MC_ReadParameter_FB.Valid THEN
	//		MC_ReadParameter_FB.Enable := FALSE;
	//		gParDataEksen12.Offset := MC_ReadParameter_FB.Value + EksenBuradaykenGormekIstedigimPozisyonDegeri;
	//	END_IF;

	//==================================================
	//		Y Eksenine home gönderelim
	//==================================================
	//isHomed geldiyse Home komutunu keselim
	IF EDGEPOS(gAxBasic[AX_HEAD_Y].IsHomed) THEN
		gAxBasic[ AX_HEAD_Y ].Home 			:= FALSE;
	END_IF;
	IF gHMI.Cmd.bHome.Ax[AX_HEAD_Y] THEN
		IF gSimulation THEN
			gAxBasicPar[AX_HEAD_Y].Homing.Mode 	:= mcHOMING_DIRECT;
			gAxBasicPar[ AX_HEAD_Y].Homing.Position	:= gFixData.Ax[AX_HEAD_Y].Par.Homing.Position;
			gAxBasic[ AX_HEAD_Y].Home 			:= gFixData.Ax[ AX_HEAD_Y].Enabled;
		ELSE
			gAxBasicPar[AX_HEAD_Y].Homing.Mode					  	:= mcHOMING_ABSOLUTE_SWITCH;
			gAxBasicPar[AX_HEAD_Y].Homing.Options.SensorOffset   	:= gFixData.Ax[AX_HEAD_Y].Config.MultiturnEncOffset; //Home yaptiktan sonra kaçinci pozisyona kadar gitsin
			gAxBasicPar[AX_HEAD_Y].Homing.Position 			  		:= gFixData.Ax[AX_HEAD_Y].Par.Homing.Position; //Home yapip Sensor offset kadar gidip bunuda üstüne ekliyor
			gAxBasicPar[AX_HEAD_Y].Homing.Options.SwitchEdge     	:= mcDIR_NEGATIVE; //Switch nerede aranacak
			gAxBasicPar[AX_HEAD_Y].Homing.Options.HomingDirection	:= mcDIR_POSITIVE; //switch ten kurtulduktan sonra offset için hangi yöne gidecek
			gAxBasicPar[AX_HEAD_Y].Homing.Options.StartDirection 	:= mcDIR_NEGATIVE;
			gAxBasicPar[AX_HEAD_Y].Homing.Options.StartVelocity  	:= 60;
			gAxBasicPar[AX_HEAD_Y].Homing.Options.HomingVelocity 	:= 30;
			gAxBasicPar[AX_HEAD_Y].Homing.Options.Acceleration   	:= 150;
			gAxBasic[AX_HEAD_Y].Home 								:= TRUE;
		END_IF;

	END_IF;

	//==================================================
	//		Vacuum Eksenine home gönderelim
	//==================================================
	//isHomed geldiyse Home komutunu keselim
	IF EDGEPOS(gAxBasic[AX_VACUUM].IsHomed) THEN
		gAxBasic[ AX_VACUUM].Home 			:= FALSE;
	END_IF;
	IF gHMI.Cmd.bHome.Ax[AX_VACUUM] THEN
		IF gSimulation THEN
			gAxBasicPar[AX_VACUUM].Homing.Mode 	:= mcHOMING_DIRECT;
			gAxBasicPar[ AX_VACUUM].Homing.Position	:= gFixData.Ax[AX_VACUUM].Par.Homing.Position;
			gAxBasic[ AX_VACUUM].Home 			:= gFixData.Ax[ AX_VACUUM].Enabled;
		ELSE
			gAxBasicPar[AX_VACUUM].Homing.Mode					  := mcHOMING_ABSOLUTE_SWITCH;
			gAxBasicPar[AX_VACUUM].Homing.Options.SensorOffset   := gFixData.Ax[AX_VACUUM].Config.MultiturnEncOffset; //Home yaptiktan sonra kaçinci pozisyona kadar gitsin
			gAxBasicPar[AX_VACUUM].Homing.Position 			  	:= gFixData.Ax[AX_VACUUM].Par.Homing.Position; //Home yapip Sensor offset kadar gidip bunuda üstüne ekliyor
			gAxBasicPar[AX_VACUUM].Homing.Options.SwitchEdge     := mcDIR_NEGATIVE; //Switch nerede aranacak
			gAxBasicPar[AX_VACUUM].Homing.Options.HomingDirection:= mcDIR_POSITIVE; //switch ten kurtulduktan sonra offset için hangi yöne gidecek
			gAxBasicPar[AX_VACUUM].Homing.Options.StartDirection := mcDIR_NEGATIVE;
			gAxBasicPar[AX_VACUUM].Homing.Options.StartVelocity  := 60;
			gAxBasicPar[AX_VACUUM].Homing.Options.HomingVelocity := 30;
			gAxBasicPar[AX_VACUUM].Homing.Options.Acceleration   := 150;
			gAxBasic[ AX_VACUUM].Home 							:= TRUE;
		END_IF;

	END_IF;

	//==================================================
	//		Köprü 1 Eksenine home gönderelim
	//==================================================
	//isHomed geldiyse Home komutunu keselim
	IF EDGEPOS(gAxBasic[AX_EXIT1_BRIDGE_Y].IsHomed) THEN
		gAxBasic[ AX_EXIT1_BRIDGE_Y].Home 			:= FALSE;
	END_IF;
	IF gHMI.Cmd.bHome.Ax[AX_EXIT1_BRIDGE_Y] THEN
		IF gSimulation THEN
			gAxBasicPar[AX_EXIT1_BRIDGE_Y].Homing.Mode 	:= mcHOMING_DIRECT;
			gAxBasicPar[ AX_EXIT1_BRIDGE_Y].Homing.Position	:= gFixData.Ax[AX_EXIT1_BRIDGE_Y].Par.Homing.Position;
			gAxBasic[ AX_EXIT1_BRIDGE_Y].Home 			:= gFixData.Ax[ AX_EXIT1_BRIDGE_Y].Enabled;
		ELSE
			gAxBasicPar[AX_EXIT1_BRIDGE_Y].Homing.Mode					  := mcHOMING_ABSOLUTE_SWITCH;
			gAxBasicPar[AX_EXIT1_BRIDGE_Y].Homing.Options.SensorOffset   := gFixData.Ax[AX_EXIT1_BRIDGE_Y].Config.MultiturnEncOffset; //Home yaptiktan sonra kaçinci pozisyona kadar gitsin
			gAxBasicPar[AX_EXIT1_BRIDGE_Y].Homing.Position 			  	:= gFixData.Ax[AX_EXIT1_BRIDGE_Y].Par.Homing.Position; //Home yapip Sensor offset kadar gidip bunuda üstüne ekliyor
			gAxBasicPar[AX_EXIT1_BRIDGE_Y].Homing.Options.SwitchEdge     := mcDIR_NEGATIVE; //Switch nerede aranacak
			gAxBasicPar[AX_EXIT1_BRIDGE_Y].Homing.Options.HomingDirection:= mcDIR_POSITIVE; //switch ten kurtulduktan sonra offset için hangi yöne gidecek
			gAxBasicPar[AX_EXIT1_BRIDGE_Y].Homing.Options.StartDirection := mcDIR_NEGATIVE;
			gAxBasicPar[AX_EXIT1_BRIDGE_Y].Homing.Options.StartVelocity  := 60;
			gAxBasicPar[AX_EXIT1_BRIDGE_Y].Homing.Options.HomingVelocity := 30;
			gAxBasicPar[AX_EXIT1_BRIDGE_Y].Homing.Options.Acceleration   := 150;
			gAxBasic[ AX_EXIT1_BRIDGE_Y].Home 							:= TRUE;
		END_IF;

	END_IF;

	//==================================================
	//		Köprü 2 Eksenine home gönderelim
	//==================================================
	IF EDGEPOS(gHMI.Cmd.bHome.Bridge[EXIT2_UNIT]) THEN
		fbExitBridgeCtrl_0[EXIT2_UNIT].In.Cmd.Home := TRUE;
		gHMI.Cmd.bHome.Bridge[EXIT2_UNIT] := FALSE;
	END_IF;

	IF EDGEPOS(gHMI.Cmd.bCalculate.Bridge[AS_BRIDGE_EXIT2]) THEN
		fbScaleBridgeExit[AS_BRIDGE_EXIT2].In.Cmd.Calculate := TRUE;
	END_IF

	fbExitBridgeCtrl_0[AS_BRIDGE_EXIT2]();
	fbScaleBridgeExit[AS_BRIDGE_EXIT2]();

	//==================================================
	//		Köprü 3 Eksenine home gönderelim
	//==================================================
	IF EDGEPOS(gHMI.Cmd.bHome.Bridge[EXIT3_UNIT]) THEN
		fbExitBridgeCtrl_0[EXIT3_UNIT].In.Cmd.Home := TRUE;
		gHMI.Cmd.bHome.Bridge[EXIT3_UNIT] := FALSE;
	END_IF;

	IF EDGEPOS(gHMI.Cmd.bCalculate.Bridge[EXIT3_UNIT]) THEN
		fbScaleBridgeExit[EXIT3_UNIT].In.Cmd.Calculate := TRUE;
	END_IF

	fbExitBridgeCtrl_0[AS_BRIDGE_EXIT3]();
	fbScaleBridgeExit[AS_BRIDGE_EXIT3]();

	//==================================================
	//		Köprü 4 Eksenine home gönderelim
	//==================================================
	IF EDGEPOS(gHMI.Cmd.bHome.Bridge[EXIT4_UNIT]) THEN
		fbExitBridgeCtrl_0[EXIT4_UNIT].In.Cmd.Home := TRUE;
		gHMI.Cmd.bHome.Bridge[EXIT4_UNIT] := FALSE;
	END_IF;

	IF EDGEPOS(gHMI.Cmd.bCalculate.Bridge[EXIT4_UNIT]) THEN
		fbScaleBridgeExit[EXIT4_UNIT].In.Cmd.Calculate := TRUE;
	END_IF

	fbExitBridgeCtrl_0[AS_BRIDGE_EXIT4]();
	fbScaleBridgeExit[AS_BRIDGE_EXIT4]();

	//==================================================
	//		Entry 1 Thickness home gönderelim
	//==================================================
	IF EDGEPOS(gHMI.Cmd.bHome.EntryThickness[ENTR1_UNIT]) THEN
		fbEntryZAscMotorCtrl[ENTR1_UNIT].In.Cmd.Home := TRUE;
		gHMI.Cmd.bHome.EntryThickness[ENTR1_UNIT] := FALSE;
	END_IF;

	IF EDGEPOS(gHMI.Cmd.bCalculate.EntryThickness[ENTR1_UNIT]) THEN
		fbScaleZAxesEntry[ENTR1_UNIT].In.Cmd.Calculate := TRUE;
	END_IF

	fbEntryZAscMotorCtrl[ENTR1_UNIT]();
	fbScaleZAxesEntry[ENTR1_UNIT]();

	//==================================================
	//		Entry 1 Thickness home gönderelim
	//==================================================
	IF EDGEPOS(gHMI.Cmd.bHome.EntryThickness[ENTR1_UNIT]) THEN
		fbEntryZAscMotorCtrl[ENTR1_UNIT].In.Cmd.Home := TRUE;
		gHMI.Cmd.bHome.EntryThickness[ENTR1_UNIT] := FALSE;
	END_IF;

	IF EDGEPOS(gHMI.Cmd.bCalculate.EntryThickness[ENTR1_UNIT]) THEN
		fbScaleZAxesEntry[ENTR1_UNIT].In.Cmd.Calculate := TRUE;
	END_IF

	fbEntryZAscMotorCtrl[ENTR1_UNIT]();
	fbScaleZAxesEntry[ENTR1_UNIT]();

	//==================================================
	//		Entry 2 Thickness home gönderelim
	//==================================================
	IF EDGEPOS(gHMI.Cmd.bHome.EntryThickness[ENTR2_UNIT]) THEN
		fbEntryZAscMotorCtrl[ENTR2_UNIT].In.Cmd.Home := TRUE;
		gHMI.Cmd.bHome.EntryThickness[ENTR2_UNIT] := FALSE;
	END_IF;

	IF EDGEPOS(gHMI.Cmd.bCalculate.EntryThickness[ENTR2_UNIT]) THEN
		fbScaleZAxesEntry[ENTR2_UNIT].In.Cmd.Calculate := TRUE;
	END_IF

	fbEntryZAscMotorCtrl[ENTR2_UNIT]();
	fbScaleZAxesEntry[ENTR2_UNIT]();

	//==================================================
	//		Exit 1 Thickness home gönderelim
	//==================================================
	IF EDGEPOS(gHMI.Cmd.bHome.ExitThickness[EXIT1_UNIT]) THEN
		fbScaleZAxesExit[EXIT1_UNIT].In.SetValue  := gHMI.Diagnosis.ExitThickness[EXIT1_UNIT].HomePos;
		fbExitZAscMotorCtrl[EXIT1_UNIT].In.Cmd.Home := TRUE;
		gHMI.Cmd.bHome.ExitThickness[EXIT1_UNIT] := FALSE;
	END_IF;

	IF EDGEPOS(gHMI.Cmd.bCalculate.ExitThickness[EXIT1_UNIT]) THEN
		fbScaleZAxesExit[EXIT1_UNIT].In.Cmd.Calculate := TRUE;
	END_IF

	fbExitZAscMotorCtrl[EXIT1_UNIT]();
	fbScaleZAxesExit[EXIT1_UNIT]();

	//==================================================
	//		Exit 2 Thickness home gönderelim
	//==================================================
	IF EDGEPOS(gHMI.Cmd.bHome.ExitThickness[EXIT2_UNIT]) THEN
		fbExitZAscMotorCtrl[EXIT2_UNIT].In.Cmd.Home := TRUE;
		gHMI.Cmd.bHome.ExitThickness[EXIT2_UNIT] := FALSE;
	END_IF;

	IF EDGEPOS(gHMI.Cmd.bCalculate.ExitThickness[EXIT2_UNIT]) THEN
		fbScaleZAxesExit[EXIT2_UNIT].In.Cmd.Calculate := TRUE;
	END_IF

	fbExitZAscMotorCtrl[EXIT2_UNIT]();
	fbScaleZAxesExit[EXIT2_UNIT]();

	//==================================================
	//		Exit 3 Thickness home gönderelim
	//==================================================
	IF EDGEPOS(gHMI.Cmd.bHome.ExitThickness[EXIT3_UNIT]) THEN
		fbExitZAscMotorCtrl[EXIT3_UNIT].In.Cmd.Home := TRUE;
		gHMI.Cmd.bHome.ExitThickness[EXIT3_UNIT] := FALSE;
	END_IF;

	IF EDGEPOS(gHMI.Cmd.bCalculate.ExitThickness[EXIT3_UNIT]) THEN
		fbScaleZAxesExit[EXIT3_UNIT].In.Cmd.Calculate := TRUE;
	END_IF

	fbExitZAscMotorCtrl[EXIT3_UNIT]();
	fbScaleZAxesExit[EXIT3_UNIT]();

	//==================================================
	//		Exit 4 Thickness home gönderelim
	//==================================================
	IF EDGEPOS(gHMI.Cmd.bHome.ExitThickness[EXIT4_UNIT]) THEN
		fbExitZAscMotorCtrl[EXIT4_UNIT].In.Cmd.Home := TRUE;
		gHMI.Cmd.bHome.ExitThickness[EXIT4_UNIT] := FALSE;
	END_IF;

	IF EDGEPOS(gHMI.Cmd.bCalculate.ExitThickness[EXIT4_UNIT]) THEN
		fbScaleZAxesExit[EXIT4_UNIT].In.Cmd.Calculate := TRUE;
	END_IF

	fbExitZAscMotorCtrl[EXIT4_UNIT]();
	fbScaleZAxesExit[EXIT4_UNIT]();

	//==================================================
	//		Edge Capture ile Y ekseni ayarlama.
	//==================================================
	CASE Loc.EdgeCaptureStep OF

		EC_WAIT_CMD:
			IF gHMI.EdgeCapture.Go THEN

				Loc.EdgeCaptureStep						 := EC_START;
				gHMI.EdgeCapture.Go					 := FALSE;
			END_IF;
		EC_START:
			IF Loc.FirstInStepEC THEN
				fbExit1BridgeEdgeCapture_0.In.Cmd.GlassEdgeCapture	 := TRUE;
			ELSE
				IF fbExit1BridgeEdgeCapture_0.Out.Status.CommandDone THEN
					fbExit1BridgeEdgeCapture_0.In.Cmd.GlassEdgeCapture		 := FALSE;
					Loc.EdgeCaptureStep										 := EC_OFSET;
				END_IF;

			END_IF;

		EC_OFSET:
			IF gHMI.EdgeCapture.Calculate THEN
				gFixData.Ax[AX_EXIT1_BRIDGE_Y].Par.Homing.Position := gFixData.Ax[AX_EXIT1_BRIDGE_Y].Par.Homing.Position - (fbExit1BridgeEdgeCapture_0.Out.GlassHeight.CapturedPos - gHMI.EdgeCapture.GlassSize);
				gHMI.EdgeCapture.Calculate 					 := FALSE;
				Loc.EdgeCaptureStep							 := EC_WAIT_CMD;
			END_IF;
			IF gCommUnit.Main.In.MachineReset THEN
				Loc.EdgeCaptureStep							 := EC_WAIT_CMD;
			END_IF;
		EC_FINISH:
	END_CASE;
	gHMI.EdgeCapture.CapturePos		 := LREAL_TO_REAL(fbExit1BridgeEdgeCapture_0.Out.GlassHeight.CapturedPos);
	IF gAxBasic[AX_HEAD_Y].MoveActive = FALSE AND gCommUnit.Main.In.MachineReset AND Loc.EdgeCaptureStep <> EC_WAIT_CMD THEN
	  Loc.EdgeCaptureStep	:= EC_WAIT_CMD;
	END_IF;
	Loc.FirstInStepEC := Loc.EdgeCaptureStep <> Loc.oldEdgeCaptureStep ;
	Loc.oldEdgeCaptureStep := Loc.EdgeCaptureStep;
END_ACTION
```

#### Distance.st
```iecst
ACTION Distance:

//	IF EDGEPOS(gHMI.Distance.FirstEdgeEntry[UP]) THEN
//	  	gFixData.Dist.Sealing.FirstEdgeEntry := gFixData.Dist.Sealing.FirstEdgeEntry + 1;
//	END_IF;
//
//	IF EDGEPOS(gHMI.Distance.FirstEdgeEntry[DOWN]) THEN
//		gFixData.Dist.Sealing.FirstEdgeEntry := gFixData.Dist.Sealing.FirstEdgeEntry - 1;
//	END_IF;

END_ACTION
```

### Program Logical/SourceCode/MachCfg (IEC)

#### Main.st
```iecst
PROGRAM _INIT
	//===========================================
	//			AXES LINKAGE
	//===========================================

	(* AX_X *)
	gAxBasic[AX_X].MpLink	   := ADR(gMpLink_AxisQX);
	gAxBasic[AX_X].Parameters  := ADR(gAxBasicPar[AX_X]);
	gAxBasic[AX_X].Enable	   := TRUE;

	(* AX_Y *)
	gAxBasic[AX_Y].MpLink	    := ADR(gMpLink_AxisQY);
	gAxBasic[AX_Y].Parameters 	:= ADR(gAxBasicPar[AX_Y]);
	gAxBasic[AX_Y].Enable	    := TRUE;

	(* AX_c *)
	gAxBasic[AX_C].MpLink	    := ADR(gMpLink_AxisVQZ);
	gAxBasic[AX_C].Parameters 	:= ADR(gAxBasicPar[AX_C]);
	gAxBasic[AX_C].Enable	    := TRUE;

END_PROGRAM

PROGRAM _CYCLIC

	gAxBasic[AX_X]();
	gAxBasic[AX_Y]();
	gAxBasic[AX_C]();
END_PROGRAM

PROGRAM _EXIT
	(* Insert code here *)

END_PROGRAM
```

### Program Logical/SourceCode/Kesim

#### Variables.var
```iecst
VAR
	fbTableUpDown_0 : fbTableUpDown;
END_VAR
```

#### Cyclic.st
```iecst
PROGRAM _CYCLIC
	(* Insert code here *)

	fbTableUpDown_0();

END_PROGRAM
```

### Package Logical/CuttingTable - Cutting table program

### Package Logical/CuttingTable/RecipeHandling - Recipe handling program

### RecipeHandling.typ - Package data types
```iecst
(********************************************************************
 * COPYRIGHT -- Bernecker + Rainer
 ********************************************************************
 * Package: RecipeHandling
 * File: RecipeHandling.typ
 * Author: blanca-gutim
 * Created: December 04, 2012
 ********************************************************************
 * Data types of package RecipeHandling
 ********************************************************************)
(**)
(*Enumeration to manage the state machine states*)

TYPE
	emu_RecipeControl_State :
		(
		C_MS_RECIPE_HAND_INIT := 0, (*Init state*)
		C_MS_RECIPE_HAND_PING, (*Send a ping command to the NETWORK device*)
		C_MS_RECIPE_HAND_SET_DEVPAR, (*Set device patrameters for linking teh device*)
		C_MS_RECIPE_HAND_LINK_DEV, (*Link file device (set the format for the String Parameter)*)
		C_MS_RECIPE_HAND_LIST, (*List of all recipes*)
		C_MS_RECIPE_HAND_WAIT_CMD, (*Wait commad state -Standstill state*)
		C_MS_RECIPE_HAND_UNLINK_DEV, (*Unlink file device*)
		C_MS_RECIPE_HAND_LOAD, (*Load recipe*)
		C_MS_RECIPE_HAND_SAVE, (*Save recipe*)
		C_MS_RECIPE_HAND_OVERWRITE, (*Overwrite recipe or not?*)
		C_MS_RECIPE_HAND_DELETE, (*Delete recipe*)
		C_MS_RECIPE_HAND_ERROR, (*General error state*)
		C_MS_RECIPE_HAND_ACK_ERROR, (*Acknowledge error state*)
		C_MS_RECIPE_HAND_NOERROR (*Error State - No error*)
		);
END_TYPE

(**)
(*========================================================================================================*)
(*Recipe handling interface type*)
(*========================================================================================================*)

TYPE
	Recipe_Ctrl_typ : 	STRUCT
		In : Recipe_Ctrl_In_typ; (*Input*)
		Out : Recipe_Ctrl_Out_typ; (*Output*)
	END_STRUCT;
END_TYPE

(*========================================================================================================*)
(*Recipe control: input sub-interface type*)
(*========================================================================================================*)

TYPE
	Recipe_Ctrl_In_typ : 	STRUCT
		Cmd : Recipe_Ctrl_In_Cmd_typ; (*Commands*)
		Par : Recipe_Ctrl_In_Par_typ; (*Parameters*)
		Stat : Recipe_Ctrl_In_Stat_typ; (*Status*)
	END_STRUCT;
END_TYPE

(*Recipe control: input commands sub-interface type*)

TYPE
	Recipe_Ctrl_In_Cmd_typ : 	STRUCT
		LoadRecipe : BOOL; (*Load recipe*)
		SaveRecipe : BOOL; (*Save recipe*)
		DeleteRecipe : BOOL; (*Delete recipe*)
		Refresh : BOOL; (*Refresh list of recipes*)
		OverwriteRecipe : BOOL; (*Overwrite recipe*)
		NotOverwriteRecipe : BOOL; (*Not overwrite recipe*)
		ErrorAcknowledge : BOOL; (*Acknowledges an error*)
	END_STRUCT;
END_TYPE

(*Recipe control: input parameters sub-interface type*)

TYPE
	Recipe_Ctrl_In_Par_typ : 	STRUCT
		RecipeName : STRING[32]; (*Recipe name*)
		RecipeIndex : UDINT; (*Index of the selected recipe into the recipe list*)
		Source : USINT; (*Sourde index for recipes*)
		Network : Recipe_Ctrl_In_Par_Net_typ; (*Network parameters when the file device is the NETWORK*)
	END_STRUCT;
END_TYPE

(*Recipe control: input network parameters sub-interface type*)

TYPE
	Recipe_Ctrl_In_Par_Net_typ : 	STRUCT
		Server : STRING[50]; (*Server where the shared directory is located*)
		Workgroup : STRING[50]; (*Workgroup*)
		DirName : STRING[50]; (*Name of the shared directory*)
		UserName : STRING[50]; (*User name*)
		Password : STRING[50]; (*Password*)
	END_STRUCT;
END_TYPE

(*Recipe control: input status sub-interface type*)

TYPE
	Recipe_Ctrl_In_Stat_typ : 	STRUCT
		FileHandling : File_Ctrl_Out_Stat_typ; (*File handling status*)
		CsvHandling : CSV_Ctrl_Out_Stat_typ; (*CSV handling status*)
	END_STRUCT;
END_TYPE

(*========================================================================================================*)
(*Recipe control: output sub-interface type*)
(*========================================================================================================*)

TYPE
	Recipe_Ctrl_Out_typ : 	STRUCT
		Cmd : Recipe_Ctrl_Out_Cmd_typ; (*Commands*)
		Par : Recipe_Ctrl_Out_Par_typ; (*Parameters*)
		Stat : Recipe_Ctrl_Out_Stat_typ; (*Status*)
	END_STRUCT;
END_TYPE

(*Recipe control: output commands sub-interface type*)

TYPE
	Recipe_Ctrl_Out_Cmd_typ : 	STRUCT
		FileHandling : File_Ctrl_In_Cmd_typ; (*File handling output commands*)
		CsvHandling : CSV_Ctrl_In_Cmd_typ; (*CSV handling output commands*)
	END_STRUCT;
END_TYPE

(*Recipe control: output commands sub-interface type*)

TYPE
	Recipe_Ctrl_Out_Par_typ : 	STRUCT
		FileHandling : File_Ctrl_In_Par_typ; (*File handling output parameters*)
		CsvHandling : CSV_Ctrl_In_Par_typ; (*CSV handling output parameters*)
	END_STRUCT;
END_TYPE

(*Recipe control: output status sub-interface type*)

TYPE
	Recipe_Ctrl_Out_Stat_typ : 	STRUCT
		MainState : DINT; (*Main state in numeric format*)
		MainState_Text : STRING[32]; (*Main state in text format*)
		NrRecipes : UDINT; (*Number of listed recipes*)
		RecipeList : ARRAY[0..C_MAX_NR_ELEMENTS_IN_DIR_MINUS1]OF STRING[260]; (*List of recipes*)
		OverwritePopUp : USINT; (*Variable to control the overwrite PopUp*)
		CmdDone : Recipe_Ctrl_In_Cmd_typ; (*Command done*)
		ReadyForCmd : BOOL; (*Variable to show that the program is ready to get a new command*)
(*		Error : Error_Type; (*Error information*)
	END_STRUCT;
END_TYPE
```

### RecipeHandling.var - Package variables
```iecst
(********************************************************************
 * COPYRIGHT -- Bernecker + Rainer
 ********************************************************************
 * Package: RecipeHandling
 * File: RecipeHandling.var
 * Author: blanca-gutim
 * Created: December 04, 2012
 ********************************************************************
 * Variables of package RecipeHandling
 ********************************************************************)
(**)
(*========================================================================================================*)
(*Program variables*)
(*========================================================================================================*)
VAR
	gRecipe_Ctrl : Recipe_Ctrl_typ := (0); (*Recipe control interface*)
END_VAR
(**)
(*========================================================================================================*)
(*Recipe handling constants*)
(*========================================================================================================*)
VAR CONSTANT
	C_MAX_BUFFER_SIZE_MINUS1 : UINT := 99; (*Maximun size of buffers minus 1 for list of files, directories and dates and times*)
	C_MAX_DEVICE_PARAM_LENGHT : UINT := 255; (*Maximun lenght of the device parameter string*)
	C_MAX_OBJECT_NAME_LENGHT : UINT := 45; (*Maximun lenght of the directory or file name*)
	C_FILE_EXTENSION_LOW : STRING[10] := '.csv'; (*File extension for the recipe handling in lower case*)
	C_FILE_EXTENSION : STRING[10] := '.CSV'; (*File extension for the recipe handling upper case (the csv file handling saves the files with this extension)*)
	C_MAX_NR_ELEMENTS_IN_DIR_MINUS1 : USINT := 99; (*Maximum number of elements in a directory*)
	C_FILE_DEVICE_CF : USINT := 0; (*Index of the CF when it is working as file device*)
	C_FILE_DEVICE_USB : USINT := 1; (*Index of the USB when it is working as file device*)
	C_FILE_DEVICE_FTP : USINT := 2; (*Index of the CF when it is working as file device*)
	C_FILE_DEVICE_NETWORK : USINT := 3; (*Index of the shared folder in the Network when it is working as file device*)
	C_GCODE_DEVICE_NETWORK : USINT := 0; (*Index of the shared folder in the Network when it is working as file device*)
	C_GCODE_DEVICE_CF : USINT := 1; (*Index of the CF when it is working as file device*)
	C_GCODE_DEVICE_USB : USINT := 2; (*Index of the USB when it is working as file device*)
	C_GCODE_DEVICE_FTP : USINT := 3; (*Index of the CF when it is working as file device*)
	C_USB_DEVICES_MAX_MINUS1 : USINT := 1; (*Maximum number of USB devices supported in the PLC minus 1*)
	C_SEPARATOR : USINT := 59; (*Separator for CSV files - ; (ASCII code of the character)*)
	C_NR_VARIABLES_CSVFILE_MINUS1 : USINT := 0; (*Number of variables that are part of the CSV file minus 1*)
	C_FILE_NAME_START : STRING[60] := 'CSV_File_'; (*Start of the file name*)
	C_SHOW_VAR_NAME_OPTION : BOOL := FALSE; (*Show the complete name of the variables (TRUE) or just a part of it (FALSE)*)
	C_MAX_LINKED_FILE_DEVICES_MINUS1 : USINT := 1; (*Maximun number of linked files devices minus 1*)
	C_PING_NETWORK_DEVICE_TIMEOUT : UINT := 500; (*Timeout for the PING command when the network device is used*)
	C_USER_DIRECTORY : STRING[10] := 'UserFiles'; (*Name for the user files in the CF*)
END_VAR
```

### Program Logical/CuttingTable/RecipeHandling/Recipe_Ctrl (IEC) - Recipe control program

#### Recipe_CtrlCyclic.st - Cyclic code
```iecst
(********************************************************************
 * COPYRIGHT -- Bernecker + Rainer
 ********************************************************************
 * PROGRAM: gRecipe_Ctrl
 * File: gRecipe_CtrlCyclic.st
 * Author: blanca-gutim
 * Created: December 04, 2012
 ********************************************************************
 * Implementation OF PROGRAM gRecipe_Ctrl
 ********************************************************************)

PROGRAM _CYCLIC

	IF uAdr <> 0 AND stat = 0 THEN
		//Update inputs
		Action_Input;

		//Control of the process if the USB is selected as File Device, but it is removed manually
		IF ( (gRecipe_Ctrl.In.Stat.FileHandling.UsbInformation[0].ifName = '') AND (gRecipe_Ctrl.In.Par.Source = C_FILE_DEVICE_USB) ) THEN
			//Change device index to CF and go to Unlink file device
			gRecipe_Ctrl.In.Par.Source 						:= C_FILE_DEVICE_CF;
		END_IF

		//Check for errors
		Action_CheckError;

		//Pop up message informing user about file operation is being executed
		//    IF (MainState = C_MS_RECIPE_HAND_DELETE OR MainState = C_MS_RECIPE_HAND_LOAD OR
		//       MainState = C_MS_RECIPE_HAND_OVERWRITE OR MainState = C_MS_RECIPE_HAND_SAVE) AND gHMI.Others.PopUpRequest = 1  THEN
		//        gHMI.Others.PopUpRequest	        	:= 0;
		//        gHMI.Others.PopUpRequestIndex                       := 207;
		//
		//    END_IF
		IF (gRecipe_Ctrl.In.Cmd.DeleteRecipe > OldInputs.Cmd.DeleteRecipe) OR (gRecipe_Ctrl.In.Cmd.LoadRecipe > OldInputs.Cmd.LoadRecipe) OR
			(gRecipe_Ctrl.In.Cmd.SaveRecipe > OldInputs.Cmd.SaveRecipe) OR (gRecipe_Ctrl.In.Cmd.Refresh > OldInputs.Cmd.Refresh)           OR
			(gRecipe_Ctrl.In.Cmd.OverwriteRecipe > OldInputs.Cmd.OverwriteRecipe)                                                          THEN
			gHMI.Others.PopUpRequestIndex := 207;
			gHMI.Others.PopUpRequest	  := 0;
			gHMI.Others.PopUpBtnCancStat  := HIDE_OBJ;
			gHMI.Others.PopUpBtnOkStat    := HIDE_OBJ;
		END_IF

		IF (gRecipe_Ctrl.Out.Stat.CmdDone.DeleteRecipe > OldOutputStatus.CmdDone.DeleteRecipe)       OR
			(gRecipe_Ctrl.Out.Stat.CmdDone.LoadRecipe > OldOutputStatus.CmdDone.LoadRecipe)           OR
			(gRecipe_Ctrl.Out.Stat.CmdDone.SaveRecipe > OldOutputStatus.CmdDone.SaveRecipe)           OR
			(gRecipe_Ctrl.Out.Stat.CmdDone.Refresh > OldOutputStatus.CmdDone.Refresh)                 OR
			(gRecipe_Ctrl.Out.Stat.CmdDone.OverwriteRecipe > OldOutputStatus.CmdDone.OverwriteRecipe) THEN
			gHMI.Others.PopUpRequestIndex := 0;
			gHMI.Others.PopUpRequest	  := 1;

		END_IF

		//====================================================================================================
		//
		//									MAIN STATE MACHINE
		//
		//====================================================================================================

		CASE MainState OF

			//============================================================================================
			C_MS_RECIPE_HAND_INIT:						//INITIALIZATION STATE
				//============================================================================================

				//TWait for the low-level task to be ready
				IF ( (gRecipe_Ctrl.In.Stat.FileHandling.ReadyForCmd = TRUE) AND (gRecipe_Ctrl.In.Stat.CsvHandling.ReadyForCmd = TRUE) ) THEN
					//Tasks ready, link the sourde file device if necessary. When there is a recover from an error is not necessary
					IF (gRecipe_Ctrl.In.Stat.FileHandling.FileDeviceInfo.FileDeviceLinked = FALSE) THEN
						//It is necessary to link the file device
						MainState 			:= C_MS_RECIPE_HAND_SET_DEVPAR;
					ELSE
						//It is not necessary to link the file device
						MainState 			:= C_MS_RECIPE_HAND_LIST;
					END_IF
				END_IF

			//============================================================================================
			C_MS_RECIPE_HAND_SET_DEVPAR:				//PREPARE STRING PARAMETER FOR SOURCE DEVICE
				//============================================================================================

				//Set the format to the Parameter string to Link the file device
				IF (gRecipe_Ctrl.Out.Cmd.FileHandling.LinkFileDevice = FALSE) AND (gRecipe_Ctrl.In.Stat.FileHandling.FileDeviceInfo.FileDeviceLinked = FALSE) THEN
					IF (gRecipe_Ctrl.In.Par.Source = C_FILE_DEVICE_CF) THEN
						//CF
						gRecipe_Ctrl.Out.Par.FileHandling.ParameterString			:= '/DEVICE=C:\\';
						gRecipe_Ctrl.Out.Par.FileHandling.DeviceName				:= 'CF';
					ELSIF (gRecipe_Ctrl.In.Par.Source = C_FILE_DEVICE_USB) THEN
						//USB
						gRecipe_Ctrl.Out.Par.FileHandling.DeviceName				:= 'USB';
						gRecipe_Ctrl.Out.Par.FileHandling.ParameterString			:= '/DEVICE=';
						strcat(ADR(gRecipe_Ctrl.Out.Par.FileHandling.ParameterString), ADR(gRecipe_Ctrl.In.Stat.FileHandling.UsbInformation[0].ifName));
					ELSIF (gRecipe_Ctrl.In.Par.Source = C_FILE_DEVICE_FTP) THEN
						//FTP
						gRecipe_Ctrl.Out.Par.FileHandling.DeviceName				:= 'FTP';
						gRecipe_Ctrl.Out.Par.FileHandling.ParameterString			:= '/PROTOCOL=ftp /SIP=';
						strcat(ADR(gRecipe_Ctrl.Out.Par.FileHandling.ParameterString), ADR(gParameters.Network.Server));
						strcat(ADR(gRecipe_Ctrl.Out.Par.FileHandling.ParameterString), ADR(' /SNAME=FTP_SERV /PROTOCOL=ftp /USER=max /PASSWORD=passw'));
					ELSIF (gRecipe_Ctrl.In.Par.Source = C_FILE_DEVICE_NETWORK) THEN
						//Network
						gRecipe_Ctrl.Out.Par.FileHandling.DeviceName				:= 'NET';
						gRecipe_Ctrl.Out.Par.FileHandling.ParameterString			:= '/PROTOCOL=cifs /SIP=';
						strcat(ADR(gRecipe_Ctrl.Out.Par.FileHandling.ParameterString), ADR(gParameters.Network.Server));
						strcat(ADR(gRecipe_Ctrl.Out.Par.FileHandling.ParameterString), ADR(' /SHARE='));
						strcat(ADR(gRecipe_Ctrl.Out.Par.FileHandling.ParameterString), ADR(gParameters.Network.DirName));
						strcat(ADR(gRecipe_Ctrl.Out.Par.FileHandling.ParameterString), ADR(' /USER='));
						strcat(ADR(gRecipe_Ctrl.Out.Par.FileHandling.ParameterString), ADR(gParameters.Network.UserName));
						strcat(ADR(gRecipe_Ctrl.Out.Par.FileHandling.ParameterString), ADR(' /PASSWORD='));
						strcat(ADR(gRecipe_Ctrl.Out.Par.FileHandling.ParameterString), ADR(gParameters.Network.Password));
						strcat(ADR(gRecipe_Ctrl.Out.Par.FileHandling.ParameterString), ADR(' /DOMAIN='));
						strcat(ADR(gRecipe_Ctrl.Out.Par.FileHandling.ParameterString), ADR(gParameters.Network.Workgroup));
					END_IF
				END_IF

				//Set next state depending on the source device. For the FTP and NETWORK a PING command is sent
				IF ( (gRecipe_Ctrl.In.Par.Source = C_FILE_DEVICE_FTP) OR (gRecipe_Ctrl.In.Par.Source = C_FILE_DEVICE_NETWORK) ) THEN
					//Send PING command
					MainState		:= C_MS_RECIPE_HAND_PING;
				ELSE
					//Link source device
					MainState		:= C_MS_RECIPE_HAND_LINK_DEV;
				END_IF

			//============================================================================================
			C_MS_RECIPE_HAND_PING:				//Send PING command to the Source device
				//============================================================================================

				//Send PING command to the network device
				IcmpPing_NetworkDevice(enable := TRUE, pHost := ADR(gRecipe_Ctrl.In.Par.Network.Server), timeout := C_PING_NETWORK_DEVICE_TIMEOUT);
				//Checking the state of the function
				IF (IcmpPing_NetworkDevice.status = ERR_OK) THEN
					//The network device was found, continue. Link file device
					MainState										:= C_MS_RECIPE_HAND_LINK_DEV;
					IcmpPing_NetworkDevice.enable 					:= FALSE;
				ELSIF (IcmpPing_NetworkDevice.status = ERR_FUB_BUSY) THEN
					//Busy, connecting to the network device
				ELSE
					//Error in function to send the PING command
					IcmpPing_NetworkDevice.enable 					:= FALSE;
					//Error, the network device is not found
					gRecipe_Ctrl.Out.Stat.Error.Number				:= UINT_TO_UDINT(IcmpPing_NetworkDevice.status);
					gRecipe_Ctrl.Out.Stat.Error.Text.Line1			:= TaskName;
					gRecipe_Ctrl.Out.Stat.Error.Text.Line2			:= StateStrings[MainState];
					ErrorState										:= MainState;
					MainState										:= C_MS_RECIPE_HAND_ERROR;
				END_IF

			//============================================================================================
			C_MS_RECIPE_HAND_LINK_DEV:			//LINK FILE DEVICE
				//============================================================================================

				//Send command to execute the action when the File handling task is ready and a File Devcie has not been previously linked
				IF ( (gRecipe_Ctrl.In.Stat.FileHandling.ReadyForCmd = TRUE) AND (gRecipe_Ctrl.In.Stat.FileHandling.FileDeviceInfo.FileDeviceLinked = FALSE) ) THEN
					//The parameter string is managed before coming to this state depending on the situation
					gRecipe_Ctrl.Out.Cmd.FileHandling.LinkFileDevice				:= TRUE;
				ELSIF (gRecipe_Ctrl.In.Stat.FileHandling.FileDeviceInfo.FileDeviceLinked = TRUE) AND (gRecipe_Ctrl.In.Stat.FileHandling.ReadyForCmd = TRUE)
					AND (gRecipe_Ctrl.In.Stat.FileHandling.CmdDone.LinkFileDevice = TRUE) THEN
					//The file device has been linked, reset command
					gRecipe_Ctrl.Out.Cmd.FileHandling.LinkFileDevice				:= FALSE;
					//Make list of recipes
					MainState														:= C_MS_RECIPE_HAND_LIST;
				END_IF

			//============================================================================================
			C_MS_RECIPE_HAND_LIST:			//GET LIST OF RECIPES
				//============================================================================================

				//Send command to execute the action when the File handling task is ready and a File Devcie has not been previously linked
				IF (gRecipe_Ctrl.In.Stat.FileHandling.ReadyForCmd = TRUE) AND (gRecipe_Ctrl.Out.Cmd.FileHandling.ReadDirectory = FALSE) THEN
					//Set parameter to read directory
					gRecipe_Ctrl.Out.Par.FileHandling.DirectoryName				:= C_USER_DIRECTORY;
					//Set command to read the directory
					gRecipe_Ctrl.Out.Cmd.FileHandling.ReadDirectory				:= TRUE;
				ELSIF (gRecipe_Ctrl.In.Stat.FileHandling.ReadyForCmd = TRUE) AND (gRecipe_Ctrl.In.Stat.FileHandling.CmdDone.ReadDirectory = TRUE) THEN
					//The directory has been read, reset command and save the information
					gRecipe_Ctrl.Out.Cmd.FileHandling.ReadDirectory				:= FALSE;
					//Save the information if there are files or directory found
					IF ( gRecipe_Ctrl.In.Stat.FileHandling.DirectoryInformation.NrFiles > 0 ) THEN
						ii	:= 0;
						memset(ADR(gRecipe_Ctrl.Out.Stat.RecipeList), 0, SIZEOF(gRecipe_Ctrl.Out.Stat.RecipeList));
						FOR kk := 0 TO (gRecipe_Ctrl.In.Stat.FileHandling.DirectoryInformation.NrFiles + gRecipe_Ctrl.In.Stat.FileHandling.DirectoryInformation.NrDirectories - 1) BY 1 DO
							//Save the recipe name indexed by kk
							memcpy(ADR(SaveFileName), ADR(gRecipe_Ctrl.In.Stat.FileHandling.DirectoryInformation.ElementsInfo[kk].Filename), SIZEOF(SaveFileName));
							//Search for the CSV extension and save only this type of files
							IF (FIND(SaveFileName, C_FILE_EXTENSION_LOW) <> 0) OR (FIND(SaveFileName, C_FILE_EXTENSION) <> 0) THEN
								//CSV file found, save name
								gRecipe_Ctrl.Out.Stat.RecipeList[ii] 			:= SaveFileName;
								ii												:= ii + 1;
							END_IF
						END_FOR
						//Update number of recipes: it will be 0 when there are not recipes
						IF (ii <> 0) THEN
							gRecipe_Ctrl.Out.Stat.NrRecipes						:= ii - 1;		//-1 because the index of the recipes will start with 0
						ELSE
							gRecipe_Ctrl.Out.Stat.NrRecipes						:= 0;
						END_IF
						//Sort the recipes by name when there are more than 1
						IF (gRecipe_Ctrl.Out.Stat.NrRecipes > 0) THEN
							Action_SortRecipes;
						END_IF
					ELSE
						//No files in the list
						memset(ADR(gRecipe_Ctrl.Out.Stat.RecipeList), 0, SIZEOF(gRecipe_Ctrl.Out.Stat.RecipeList));
					END_IF
					//Go to wait command state
					gHMI.Others.PopUpRequest := HIDE_OBJ;
					MainState				 := C_MS_RECIPE_HAND_WAIT_CMD;
					//Check if the Refresh command was used or not
					IF (gRecipe_Ctrl.In.Cmd.Refresh = TRUE) THEN
						//Set Refresh output command done
						gRecipe_Ctrl.Out.Stat.CmdDone.Refresh					:= TRUE;
					END_IF
				END_IF

			//============================================================================================
			C_MS_RECIPE_HAND_WAIT_CMD:					//READY STATE
				//============================================================================================

				//WAIT FOR COMMANDS
				IF (gRecipe_Ctrl.Out.Stat.ReadyForCmd = TRUE) THEN
					IF (gRecipe_Ctrl.In.Cmd.DeleteRecipe > OldInputs.Cmd.DeleteRecipe) THEN
						//Go to Delete recipe state
						MainState			:= C_MS_RECIPE_HAND_DELETE;
					ELSIF (gRecipe_Ctrl.In.Cmd.LoadRecipe > OldInputs.Cmd.LoadRecipe) THEN
						//Go to Load Recipe state
						MainState			:= C_MS_RECIPE_HAND_LOAD;
					ELSIF (gRecipe_Ctrl.In.Cmd.SaveRecipe > OldInputs.Cmd.SaveRecipe) THEN
						IF (gRecipe_Ctrl.In.Par.RecipeName = '') THEN
							gRecipe_Ctrl.In.Par.RecipeName := gRecipe_Ctrl.Out.Stat.RecipeList[gRecipe_Ctrl.In.Par.RecipeIndex];
						END_IF;
						//Go to Save Recipe state
						MainState			:= C_MS_RECIPE_HAND_SAVE;
					ELSIF (gRecipe_Ctrl.In.Cmd.Refresh > OldInputs.Cmd.Refresh) THEN
						//Go to Refresh Recipe list state
						MainState			:= C_MS_RECIPE_HAND_LIST;
					ELSE
						//Stay in Wait Command state
						MainState 			:= C_MS_RECIPE_HAND_WAIT_CMD;
						//Reset input commands
						memset(ADR(gRecipe_Ctrl.In.Cmd), 0, SIZEOF(gRecipe_Ctrl.In.Cmd));
					END_IF
				END_IF

				//CHECK IF THE SOURCE FILE DEVICE CHANGED
				IF (gRecipe_Ctrl.In.Par.Source <> OldInputs.Par.Source) THEN
					//The selected source device changed, unlnk the actual file device and link the new one
					MainState 				:= C_MS_RECIPE_HAND_UNLINK_DEV;
				END_IF

				//Update the output ReadyForCmd
				IF (MainState = C_MS_RECIPE_HAND_WAIT_CMD) AND (gRecipe_Ctrl.In.Stat.FileHandling.ReadyForCmd = TRUE) AND (gRecipe_Ctrl.In.Stat.CsvHandling.ReadyForCmd = TRUE) THEN
					gRecipe_Ctrl.Out.Stat.ReadyForCmd	:= TRUE;
				ELSE
					gRecipe_Ctrl.Out.Stat.ReadyForCmd	:= FALSE;
				END_IF

			//============================================================================================
			C_MS_RECIPE_HAND_UNLINK_DEV:			//UNLINK FILE DEVICE
				//============================================================================================

				//Send command to execute the action when the File handling task is ready and a File Devcie has been previously linked
				IF ( (gRecipe_Ctrl.In.Stat.FileHandling.ReadyForCmd = TRUE) AND (gRecipe_Ctrl.In.Stat.FileHandling.FileDeviceInfo.FileDeviceLinked = TRUE) ) THEN
					//The parameter string is managed before coming to this state depending on the situation
					gRecipe_Ctrl.Out.Cmd.FileHandling.UnlinkFileDevice			:= TRUE;
				ELSIF (gRecipe_Ctrl.In.Stat.FileHandling.FileDeviceInfo.FileDeviceLinked = FALSE) AND (gRecipe_Ctrl.In.Stat.FileHandling.ReadyForCmd = TRUE)
					AND (gRecipe_Ctrl.In.Stat.FileHandling.CmdDone.UnlinkFileDevice = TRUE) THEN
					//The file device has been unlinked, reset command
					gRecipe_Ctrl.Out.Cmd.FileHandling.UnlinkFileDevice			:= FALSE;
					//Link the new file device
					MainState													:= C_MS_RECIPE_HAND_SET_DEVPAR;
				END_IF

			//============================================================================================
			C_MS_RECIPE_HAND_DELETE:			//DELETE RECIPE
				//============================================================================================

				//Send command to execute the action when the File handling task is ready and a recipe is selected
				IF ( (gRecipe_Ctrl.In.Stat.FileHandling.ReadyForCmd = TRUE) AND (gRecipe_Ctrl.Out.Stat.RecipeList[gRecipe_Ctrl.In.Par.RecipeIndex] <> '') AND
					(gRecipe_Ctrl.Out.Cmd.FileHandling.DeleteFile = FALSE) ) THEN
					//Set command and parameters to delete file
					gRecipe_Ctrl.Out.Par.FileHandling.FileName					:= C_USER_DIRECTORY;
					strcat(ADR(gRecipe_Ctrl.Out.Par.FileHandling.FileName), ADR('/'));
					strcat(ADR(gRecipe_Ctrl.Out.Par.FileHandling.FileName), ADR(gRecipe_Ctrl.Out.Stat.RecipeList[gRecipe_Ctrl.In.Par.RecipeIndex]));
					gRecipe_Ctrl.Out.Cmd.FileHandling.DeleteFile				:= TRUE;
				ELSIF (gRecipe_Ctrl.In.Stat.FileHandling.CmdDone.DeleteFile = TRUE) AND (gRecipe_Ctrl.In.Stat.FileHandling.ReadyForCmd = TRUE)
					AND (gRecipe_Ctrl.Out.Cmd.FileHandling.DeleteFile = TRUE) THEN
					//The recipe has been deleted, reset command
					gRecipe_Ctrl.Out.Cmd.FileHandling.DeleteFile				:= FALSE;
					//Set output command done
					gRecipe_Ctrl.Out.Stat.CmdDone.DeleteRecipe					:= TRUE;
					//Make again the list of files
					MainState													:= C_MS_RECIPE_HAND_LIST;
				ELSIF (gRecipe_Ctrl.Out.Stat.RecipeList[gRecipe_Ctrl.In.Par.RecipeIndex] = '') THEN
					//No file selected, go back to wait command
					gHMI.Others.PopUpRequest	        	                        := 1;
					MainState													:= C_MS_RECIPE_HAND_WAIT_CMD;
				END_IF

			//============================================================================================
			C_MS_RECIPE_HAND_SAVE:			//SAVE RECIPE
				//============================================================================================

				//Send command to execute the action when the File handling task is ready and a recipe is selected
				IF ( (gRecipe_Ctrl.In.Stat.FileHandling.ReadyForCmd = TRUE) AND (gRecipe_Ctrl.In.Par.RecipeName <> '') AND
					(gRecipe_Ctrl.Out.Cmd.CsvHandling.WriteFile = FALSE) ) THEN
					//Set command and parameters to save file
					gRecipe_Ctrl.Out.Par.CsvHandling.FileDeviceName	:= gRecipe_Ctrl.In.Stat.FileHandling.FileDeviceInfo.Name;
					gRecipe_Ctrl.Out.Par.CsvHandling.FileName		:= gRecipe_Ctrl.In.Par.RecipeName;
					gRecipe_Ctrl.Out.Par.CsvHandling.Path			:= C_USER_DIRECTORY;
					strcat(ADR(gRecipe_Ctrl.Out.Par.CsvHandling.Path), ADR('\'));
					gRecipe_Ctrl.Out.Cmd.CsvHandling.WriteFile		:= TRUE;
				ELSIF (gRecipe_Ctrl.In.Stat.CsvHandling.CmdDone.WriteFile = TRUE) AND (gRecipe_Ctrl.In.Stat.FileHandling.ReadyForCmd = TRUE)
					AND (gRecipe_Ctrl.Out.Cmd.CsvHandling.WriteFile = TRUE) THEN
					//The recipe has been saved, reset command
					gRecipe_Ctrl.Out.Cmd.CsvHandling.WriteFile		:= FALSE;
					//Set output command done
					gRecipe_Ctrl.Out.Stat.CmdDone.SaveRecipe		:= TRUE;
					//Make again the list of files
					MainState										:= C_MS_RECIPE_HAND_LIST;
				ELSIF (gRecipe_Ctrl.Out.Cmd.CsvHandling.WriteFile = TRUE) AND (gRecipe_Ctrl.In.Stat.CsvHandling.FileAlreadyExists = TRUE) THEN
					//There is already a file with the same name, overwrite or not
					//Reset pop up
					gHMI.Others.PopUpRequest	        	:= 0;
					gHMI.Others.PopUpRequestIndex           := 217;
					gHMI.Others.PopUpBtnCancStat            := SHOW_OBJ;
					gHMI.Others.PopUpBtnOkStat              := SHOW_OBJ;
					MainState								:= C_MS_RECIPE_HAND_OVERWRITE;
				ELSIF (gRecipe_Ctrl.In.Par.RecipeName = '') THEN
					//No recipe name entered, go back to wait command
					gRecipe_Ctrl.In.Par.RecipeName := gRecipe_Ctrl.Out.Stat.RecipeList[gRecipe_Ctrl.In.Par.RecipeIndex];
				END_IF

			//============================================================================================
			C_MS_RECIPE_HAND_OVERWRITE:			//OVERWRITE RECIPE OR NOT
				//============================================================================================
				IF gHMI.Others.PopUpRequest = SHOW_OBJ THEN
					IF gHMI.Others.CmdOk THEN
						gHMI.Others.CmdOk             := FALSE;
						gHMI.Others.PopUpRequest      := SHOW_OBJ;
						gHMI.Others.PopUpBtnCancStat  := HIDE_OBJ;
						gHMI.Others.PopUpBtnOkStat    := HIDE_OBJ;
						gHMI.Others.PopUpRequestIndex := 207;
						gRecipe_Ctrl.In.Cmd.OverwriteRecipe := TRUE;
					ELSIF gHMI.Others.CmdCancel THEN
						gHMI.Others.CmdCancel := FALSE;
						gHMI.Others.CmdOk             := FALSE;
						gHMI.Others.PopUpRequest      := SHOW_OBJ;
						gRecipe_Ctrl.In.Cmd.NotOverwriteRecipe := TRUE;
					END_IF;
				END_IF;

				//Wait for user command to select if the recipe is going to be overwritten or not
				IF (gRecipe_Ctrl.Out.Cmd.CsvHandling.OverwriteFile = FALSE) AND (gRecipe_Ctrl.Out.Cmd.CsvHandling.NotOverwriteFile = FALSE) THEN
					IF (gRecipe_Ctrl.In.Cmd.OverwriteRecipe > OldInputs.Cmd.OverwriteRecipe) THEN
						//Overwrite recipe, send command to CSV handling task
						gRecipe_Ctrl.Out.Cmd.CsvHandling.OverwriteFile		:= TRUE;
					ELSIF (gRecipe_Ctrl.In.Cmd.NotOverwriteRecipe > OldInputs.Cmd.NotOverwriteRecipe) THEN
						//Not overwrite recipe, send command to CSV handling task
						gRecipe_Ctrl.Out.Cmd.CsvHandling.NotOverwriteFile	:= TRUE;
					END_IF
				END_IF
				//Wait for the process to be finished
				IF ( (gRecipe_Ctrl.Out.Cmd.CsvHandling.OverwriteFile = TRUE) OR (gRecipe_Ctrl.Out.Cmd.CsvHandling.NotOverwriteFile = TRUE) ) AND
					(gRecipe_Ctrl.In.Stat.CsvHandling.ReadyForCmd = TRUE) THEN
					IF (gRecipe_Ctrl.In.Stat.CsvHandling.CmdDone.OverwriteFile = TRUE) AND (gRecipe_Ctrl.In.Stat.CsvHandling.CmdDone.WriteFile = TRUE) THEN
						//Reset command
						gRecipe_Ctrl.Out.Cmd.CsvHandling.OverwriteFile		:= FALSE;
						//Set output command done
						gRecipe_Ctrl.Out.Stat.CmdDone.OverwriteRecipe		:= TRUE;
					ELSIF (gRecipe_Ctrl.In.Stat.CsvHandling.CmdDone.NotOverwriteFile = TRUE) AND (gRecipe_Ctrl.In.Stat.CsvHandling.CmdDone.WriteFile = TRUE) THEN
						//Reset command
						gRecipe_Ctrl.Out.Cmd.CsvHandling.NotOverwriteFile	:= FALSE;
						//Set output command done
						gRecipe_Ctrl.Out.Stat.CmdDone.NotOverwriteRecipe	:= TRUE;
					END_IF
					//Reset write file command
					gRecipe_Ctrl.Out.Cmd.CsvHandling.WriteFile				:= FALSE;
					//Set output command done
					gRecipe_Ctrl.Out.Stat.CmdDone.SaveRecipe				:= TRUE;
					//Go to wait command state
					gHMI.Others.PopUpRequest	        	                := 1;
					gHMI.Others.PopUpRequestIndex                           := 0;
					MainState												:= C_MS_RECIPE_HAND_WAIT_CMD;
				END_IF

			//============================================================================================
			C_MS_RECIPE_HAND_LOAD:			//LOAD RECIPE
				//============================================================================================

				//Send command to execute the action when the File handling task is ready and a recipe is selected
				IF ( (gRecipe_Ctrl.In.Stat.FileHandling.ReadyForCmd = TRUE) AND (gRecipe_Ctrl.Out.Stat.RecipeList[gRecipe_Ctrl.In.Par.RecipeIndex] <> '') AND
					(gRecipe_Ctrl.Out.Cmd.CsvHandling.ReadFile = FALSE) ) THEN
					//Set command and parameters to load file
					gRecipe_Ctrl.Out.Par.CsvHandling.FileDeviceName				:= gRecipe_Ctrl.In.Stat.FileHandling.FileDeviceInfo.Name;
					gRecipe_Ctrl.Out.Par.CsvHandling.FileName					:= gRecipe_Ctrl.Out.Stat.RecipeList[gRecipe_Ctrl.In.Par.RecipeIndex];
					gRecipe_Ctrl.Out.Par.CsvHandling.Path						:= C_USER_DIRECTORY;
					strcat(ADR(gRecipe_Ctrl.Out.Par.CsvHandling.Path), ADR('\'));
					gRecipe_Ctrl.Out.Cmd.CsvHandling.ReadFile					:= TRUE;
				ELSIF (gRecipe_Ctrl.In.Stat.CsvHandling.CmdDone.ReadFile = TRUE) AND (gRecipe_Ctrl.In.Stat.FileHandling.ReadyForCmd = TRUE)
					AND (gRecipe_Ctrl.Out.Cmd.CsvHandling.ReadFile = TRUE) THEN
					//The recipe has been loaded, reset command
					gRecipe_Ctrl.Out.Cmd.CsvHandling.ReadFile					:= FALSE;
					//Set output command done
					gRecipe_Ctrl.Out.Stat.CmdDone.LoadRecipe					:= TRUE;
					pAuto_Ctrl.In.Stat.RecipeLoaded                             := TRUE;
					//Go to wait command state
					gHMI.Others.PopUpRequest	        	                    := 1;
					gRecipe_Ctrl.In.Par.RecipeName                              := '';
					MainState													:= C_MS_RECIPE_HAND_WAIT_CMD;
					//Copy gloabal parameters structure to local loader parameters to
					gLoaderControl.In.Par										:= gParameters.LoaderParameters;
				ELSIF (gRecipe_Ctrl.Out.Stat.RecipeList[gRecipe_Ctrl.In.Par.RecipeIndex] = '') THEN
					//No recipe selected, go back to wait command
					gHMI.Others.PopUpRequest	        	                    := 1;
					MainState													:= C_MS_RECIPE_HAND_WAIT_CMD;
				END_IF

			//============================================================================================
			C_MS_RECIPE_HAND_ERROR:				//ERROR HANDLING
				//============================================================================================

				gHMI.Others.PopUpRequest	        	                        := 1;
				//Wait for user acknowledge
				IF (gRecipe_Ctrl.In.Cmd.ErrorAcknowledge > OldInputs.Cmd.ErrorAcknowledge) THEN
					//The user wants to acknowledge the error -> Next step: Go to Acknowledge Error State
					MainState 			:= C_MS_RECIPE_HAND_ACK_ERROR;
					//Reset output commands
					memset(ADR(gRecipe_Ctrl.Out.Cmd), 0, SIZEOF(gRecipe_Ctrl.Out.Cmd));
					//Reset input commands
					memset(ADR(gRecipe_Ctrl.In.Cmd), 0, SIZEOF(gRecipe_Ctrl.In.Cmd));
				END_IF

			//============================================================================================
			C_MS_RECIPE_HAND_ACK_ERROR:			//ACKNOWLEDGE ERROR
				//============================================================================================

				//Clear error information
				gRecipe_Ctrl.Out.Stat.Error.Number							:= 0;
				memset(ADR(gRecipe_Ctrl.Out.Stat.Error.Text), 0, SIZEOF(gRecipe_Ctrl.Out.Stat.Error.Text));
				//Send acknowledge error command to the low level tasks in case that they are in error
				IF (gRecipe_Ctrl.In.Stat.FileHandling.Error.Number <> 0) THEN
					//Error in low level task, acknowledge error
					gRecipe_Ctrl.Out.Cmd.FileHandling.ErrorAcknowledge		:= TRUE;
				ELSIF ( (gRecipe_Ctrl.In.Stat.FileHandling.Error.Number = 0) AND (gRecipe_Ctrl.In.Stat.FileHandling.CmdDone.ErrorAcknowledge = TRUE) ) THEN
					//Reset output command to acknowledge
					gRecipe_Ctrl.Out.Cmd.FileHandling.ErrorAcknowledge		:= FALSE;
				END_IF
				IF (gRecipe_Ctrl.In.Stat.CsvHandling.Error.Number <> 0) THEN
					//Error in low level task, acknowledge error
					gRecipe_Ctrl.Out.Cmd.CsvHandling.ErrorAcknowledge		:= TRUE;
				ELSIF ( (gRecipe_Ctrl.In.Stat.CsvHandling.Error.Number = 0) AND (gRecipe_Ctrl.In.Stat.CsvHandling.CmdDone.ErrorAcknowledge = TRUE) ) THEN
					//Reset output command to acknowledge
					gRecipe_Ctrl.Out.Cmd.CsvHandling.ErrorAcknowledge		:= FALSE;
				END_IF
				//Check if all error numbers are 0 to set command done output status
				IF ( (gRecipe_Ctrl.In.Stat.CsvHandling.Error.Number = 0) AND (gRecipe_Ctrl.In.Stat.FileHandling.Error.Number = 0) AND (gRecipe_Ctrl.Out.Stat.Error.Number = 0) ) THEN
					//Error acknowledged
					gRecipe_Ctrl.Out.Stat.CmdDone.ErrorAcknowledge			:= TRUE;
					//Acknowledge done -> Next step: Go to Init State
					MainState 												:= C_MS_RECIPE_HAND_INIT;
					ErrorState												:= C_MS_RECIPE_HAND_NOERROR;
				END_IF

			ELSE

				//============================================================================================

				//The program sould not come here
				MainState 									:= C_MS_RECIPE_HAND_ERROR;
				gRecipe_Ctrl.Out.Stat.Error.Number			:= 0;
				gRecipe_Ctrl.Out.Stat.Error.Text.Line1		:= TaskName;
				gRecipe_Ctrl.Out.Stat.Error.Text.Line2		:= 'Not defined state in state machine';
				ErrorState									:= MainState;
				MainState									:= C_MS_RECIPE_HAND_ERROR;

			//============================================================================================

		END_CASE

		//Update variables used to detect edges
		OldInputs		:= gRecipe_Ctrl.In;
		OldOutputStatus	:= gRecipe_Ctrl.Out.Stat;
		//Update outputs
		Action_Output;

	END_IF;

END_PROGRAM
```

#### Recipe_CtrlInit.st - Initialization code
```iecst
(********************************************************************
 * COPYRIGHT -- Bernecker + Rainer
 ********************************************************************
 * PROGRAM: gRecipe_Ctrl
 * File: gRecipe_CtrlInit.st
 * Author: blanca-gutim
 * Created: December 04, 2012
 ********************************************************************
 * Implementation OF PROGRAM gRecipe_Ctrl
 ********************************************************************)

PROGRAM _INIT

	//Init of task name
	TaskName	:= 'Recipe_Ctrl';

	//Init of variables used to control state machines
	MainState	:= C_MS_RECIPE_HAND_INIT;
	ErrorState	:= C_MS_RECIPE_HAND_NOERROR;

	//Init of other variables
	gRecipe_Ctrl.In.Par.Source		:= C_FILE_DEVICE_CF;		//CF used as default source device

	//Copy gloabal parameters structure to local loader parameters to
	gLoaderControl.In.Par			:= gParameters.LoaderParameters;

	//Set the format to the Parameter string to Link the file device
	IF (gRecipe_Ctrl.In.Par.Source = C_FILE_DEVICE_CF) THEN
		//CF
		gRecipe_Ctrl.Out.Par.FileHandling.ParameterString			:= '/DEVICE=C:\\';
		gRecipe_Ctrl.Out.Par.FileHandling.DeviceName				:= 'CF';
	ELSIF (gRecipe_Ctrl.In.Par.Source = C_FILE_DEVICE_USB) THEN
		//USB
		gRecipe_Ctrl.Out.Par.FileHandling.DeviceName				:= 'USB';
		gRecipe_Ctrl.Out.Par.FileHandling.ParameterString			:= '/DEVICE=';
		strcat(ADR(gRecipe_Ctrl.Out.Par.FileHandling.ParameterString), ADR(gRecipe_Ctrl.In.Stat.FileHandling.UsbInformation[0].ifName));
	ELSIF (gRecipe_Ctrl.In.Par.Source = C_FILE_DEVICE_FTP) THEN
		//FTP
		gRecipe_Ctrl.Out.Par.FileHandling.DeviceName				:= 'FTP';
		gRecipe_Ctrl.Out.Par.FileHandling.ParameterString			:= '/PROTOCOL=ftp /SIP=';
		strcat(ADR(gRecipe_Ctrl.Out.Par.FileHandling.ParameterString), ADR(gParameters.Network.Server));
		strcat(ADR(gRecipe_Ctrl.Out.Par.FileHandling.ParameterString), ADR(' /SNAME=FTP_SERV /PROTOCOL=ftp /USER=max /PASSWORD=passw'));
	ELSIF (gRecipe_Ctrl.In.Par.Source = C_FILE_DEVICE_NETWORK) THEN
		//Network
		gRecipe_Ctrl.Out.Par.FileHandling.DeviceName				:= 'NET';
		gRecipe_Ctrl.Out.Par.FileHandling.ParameterString			:= '/PROTOCOL=cifs /SIP=';
		strcat(ADR(gRecipe_Ctrl.Out.Par.FileHandling.ParameterString), ADR(gParameters.Network.Server));
		strcat(ADR(gRecipe_Ctrl.Out.Par.FileHandling.ParameterString), ADR(' /SHARE='));
		strcat(ADR(gRecipe_Ctrl.Out.Par.FileHandling.ParameterString), ADR(gParameters.Network.DirName));
		strcat(ADR(gRecipe_Ctrl.Out.Par.FileHandling.ParameterString), ADR(' /USER='));
		strcat(ADR(gRecipe_Ctrl.Out.Par.FileHandling.ParameterString), ADR(gParameters.Network.UserName));
		strcat(ADR(gRecipe_Ctrl.Out.Par.FileHandling.ParameterString), ADR(' /PASSWORD='));
		strcat(ADR(gRecipe_Ctrl.Out.Par.FileHandling.ParameterString), ADR(gParameters.Network.Password));
		strcat(ADR(gRecipe_Ctrl.Out.Par.FileHandling.ParameterString), ADR(' /DOMAIN='));
		strcat(ADR(gRecipe_Ctrl.Out.Par.FileHandling.ParameterString), ADR(gParameters.Network.Workgroup));
	END_IF

	//Init of variable to get state names in text format
	StateStrings[C_MS_RECIPE_HAND_INIT]				:= 'C_MS_RECIPE_HAND_INIT';
	StateStrings[C_MS_RECIPE_HAND_WAIT_CMD]			:= 'C_MS_RECIPE_HAND_WAIT_CMD';
	StateStrings[C_MS_RECIPE_HAND_PING]				:= 'C_MS_RECIPE_HAND_PING';
	StateStrings[C_MS_RECIPE_HAND_SET_DEVPAR]		:= 'C_MS_RECIPE_HAND_SET_DEVPAR';
	StateStrings[C_MS_RECIPE_HAND_LINK_DEV]			:= 'C_MS_RECIPE_HAND_LINK_DEV';
	StateStrings[C_MS_RECIPE_HAND_LIST]				:= 'C_MS_RECIPE_HAND_LIST';
	StateStrings[C_MS_RECIPE_HAND_UNLINK_DEV]		:= 'C_MS_RECIPE_HAND_UNLINK_DEV';
	StateStrings[C_MS_RECIPE_HAND_LOAD]				:= 'C_MS_RECIPE_HAND_LOAD';
	StateStrings[C_MS_RECIPE_HAND_OVERWRITE]		:= 'C_MS_RECIPE_HAND_OVERWRITE';
	StateStrings[C_MS_RECIPE_HAND_SAVE]				:= 'C_MS_RECIPE_HAND_SAVE';
	StateStrings[C_MS_RECIPE_HAND_DELETE]			:= 'C_MS_RECIPE_HAND_DELETE';
	StateStrings[C_MS_RECIPE_HAND_ERROR]			:= 'C_MS_RECIPE_HAND_ERROR';
	StateStrings[C_MS_RECIPE_HAND_ACK_ERROR]		:= 'C_MS_RECIPE_HAND_ACK_ERROR';
	StateStrings[C_MS_RECIPE_HAND_NOERROR]			:= 'C_MS_RECIPE_HAND_NOERROR';

	// ----------------------------
	// Access to Program Interfaces
	// ----------------------------
	// Access to Auto_Ctrl task interface
	uAdr := 0; uSize := 0;
	stat := PV_xgetadr(ADR('Auto_Ctrl:Auto_Ctrl'), ADR(uAdr), ADR(uSize));
	IF uAdr <> 0 AND stat = 0 THEN
		pAuto_Ctrl ACCESS uAdr;
	END_IF
END_PROGRAM
```

#### Recipe_Ctrl.var - Local variables
```iecst
(********************************************************************
 * COPYRIGHT -- Bernecker + Rainer
 ********************************************************************
 * Program: Recipe_Ctrl
 * File: Recipe_Ctrl.var
 * Author: blanca-gutim
 * Created: December 04, 2012
 ********************************************************************
 * Local variables of program Recipe_Ctrl
 ********************************************************************)
VAR
	pAuto_Ctrl : REFERENCE TO Auto_Ctrl_typ;
END_VAR
(**)
(*================================================
Program variables
================================================*)
VAR
	uAdr : UDINT := 0;
	uSize : UDINT := 0;
	stat : UINT := 0;
	TaskName : STRING[20]; (*Name of the actual task, used for error handling*)
	StateStrings : ARRAY[0..15] OF STRING[32]; (*Array with the names of the possible states (update if the number of states is increased)*)
	OldInputs : Recipe_Ctrl_In_typ; (*Variable used to detect edges in the inputs*)
	OldOutputStatus : Recipe_Ctrl_Out_Stat_typ; (*Variable used to detect edges in the output status*)
	MainState : emu_RecipeControl_State; (*Main state for the control of the state machine*)
	ErrorState : emu_RecipeControl_State; (*Variable used to identify in wich state an error occurs*)
	IcmpPing_NetworkDevice : IcmpPing; (*FUB: Send a PING command to the network device*)
	SaveFileName : STRING[C_MAX_OBJECT_NAME_LENGHT]; (*Auxiliar variable used to store the name of recipes during the sorting procedure*)
	Changed : BOOL; (*Variable to control the sorting procedure of the recipes*)
	ii : UDINT; (*Variable used as counter in FOR loops*)
	kk : UDINT; (*Variable used as counter in FOR loops*)
END_VAR
```

#### Actions.st
```iecst
(********************************************************************
 * COPYRIGHT -- Bernecker + Rainer
 ********************************************************************
 * Program: gRecipe_Ctrl
 * File: Actions.st
 * Author: blanca-gutim
 * Created: December 04, 2012
 ********************************************************************
 * Implementation of program gRecipe_Ctrl
 ********************************************************************)

(* Input actions *)
ACTION Action_Input:

	//Update inputs
	gRecipe_Ctrl.In.Stat.FileHandling	:= gFile_Ctrl.Out.Stat;
	gRecipe_Ctrl.In.Stat.CsvHandling	:= gCSV_Ctrl.Out.Stat;

	//Copy local loader parameters to gloabal parameters structure
	IF (MainState = C_MS_RECIPE_HAND_WAIT_CMD) THEN
		gParameters.LoaderParameters	:= gLoaderControl.In.Par;
	END_IF

END_ACTION

(* Output actions *)
ACTION Action_Output:

	//Reset input commands when they are done
	IF (gRecipe_Ctrl.Out.Stat.CmdDone.DeleteRecipe = TRUE) THEN
		gRecipe_Ctrl.In.Cmd.DeleteRecipe			:= FALSE;
	END_IF
	IF (gRecipe_Ctrl.Out.Stat.CmdDone.ErrorAcknowledge = TRUE) THEN
		gRecipe_Ctrl.In.Cmd.ErrorAcknowledge		:= FALSE;
	END_IF
	IF (gRecipe_Ctrl.Out.Stat.CmdDone.LoadRecipe = TRUE) THEN
		gRecipe_Ctrl.In.Cmd.LoadRecipe				:= FALSE;
	END_IF
	IF (gRecipe_Ctrl.Out.Stat.CmdDone.SaveRecipe = TRUE) THEN
		gRecipe_Ctrl.In.Cmd.SaveRecipe				:= FALSE;
	END_IF
	IF (gRecipe_Ctrl.Out.Stat.CmdDone.Refresh = TRUE) THEN
		gRecipe_Ctrl.In.Cmd.Refresh					:= FALSE;
	END_IF
	IF (gRecipe_Ctrl.Out.Stat.CmdDone.OverwriteRecipe = TRUE) THEN
		gRecipe_Ctrl.In.Cmd.OverwriteRecipe			:= FALSE;
	END_IF
	IF (gRecipe_Ctrl.Out.Stat.CmdDone.NotOverwriteRecipe = TRUE) THEN
		gRecipe_Ctrl.In.Cmd.NotOverwriteRecipe		:= FALSE;
	END_IF

	//Update outputs, reset command done status
	gRecipe_Ctrl.Out.Stat.CmdDone.DeleteRecipe			:= gRecipe_Ctrl.Out.Stat.CmdDone.DeleteRecipe		AND gRecipe_Ctrl.In.Cmd.DeleteRecipe;
	gRecipe_Ctrl.Out.Stat.CmdDone.ErrorAcknowledge		:= gRecipe_Ctrl.Out.Stat.CmdDone.ErrorAcknowledge	AND gRecipe_Ctrl.In.Cmd.ErrorAcknowledge;
	gRecipe_Ctrl.Out.Stat.CmdDone.LoadRecipe			:= gRecipe_Ctrl.Out.Stat.CmdDone.LoadRecipe			AND gRecipe_Ctrl.In.Cmd.LoadRecipe;
	gRecipe_Ctrl.Out.Stat.CmdDone.SaveRecipe			:= gRecipe_Ctrl.Out.Stat.CmdDone.SaveRecipe			AND gRecipe_Ctrl.In.Cmd.SaveRecipe;
	gRecipe_Ctrl.Out.Stat.CmdDone.Refresh				:= gRecipe_Ctrl.Out.Stat.CmdDone.Refresh			AND gRecipe_Ctrl.In.Cmd.Refresh;
	gRecipe_Ctrl.Out.Stat.CmdDone.OverwriteRecipe		:= gRecipe_Ctrl.Out.Stat.CmdDone.OverwriteRecipe	AND gRecipe_Ctrl.In.Cmd.OverwriteRecipe;
	gRecipe_Ctrl.Out.Stat.CmdDone.NotOverwriteRecipe	:= gRecipe_Ctrl.Out.Stat.CmdDone.NotOverwriteRecipe	AND gRecipe_Ctrl.In.Cmd.NotOverwriteRecipe;

	//Update output, get MainState and Error State in String and UDINT variables (for tracing and debuging)
	gRecipe_Ctrl.Out.Stat.MainState						:= MainState;
	gRecipe_Ctrl.Out.Stat.MainState_Text				:= StateStrings[MainState];

	//Update network parameters for file handling task
	gRecipe_Ctrl.In.Par.Network							:= gParameters.Network;

	//Update the signal to know that the selected file already exists
	IF (MainState = C_MS_RECIPE_HAND_OVERWRITE) THEN
		//File already exists
		gRecipe_Ctrl.Out.Stat.OverwritePopUp		:= 0;
	ELSE
		//File doesn´t exists
		gRecipe_Ctrl.Out.Stat.OverwritePopUp		:= 1;
	END_IF

END_ACTION

(*Sorting procedure for recipes*)
ACTION Action_SortRecipes:

	//Sorting procedure, when recipes are found
	IF (gRecipe_Ctrl.Out.Stat.RecipeList[0] <> '') THEN
		Changed	:= FALSE;
		kk		:= 0;
		REPEAT
			IF (strcmp(ADR(gRecipe_Ctrl.Out.Stat.RecipeList[kk]),ADR(gRecipe_Ctrl.Out.Stat.RecipeList[kk+1])) > 0) AND
				(gRecipe_Ctrl.Out.Stat.RecipeList[kk] <> '') AND (gRecipe_Ctrl.Out.Stat.RecipeList[kk+1] <> '') THEN
				Changed := TRUE;
				strcpy(ADR(SaveFileName), ADR(gRecipe_Ctrl.Out.Stat.RecipeList[kk+1]));
				strcpy(ADR(gRecipe_Ctrl.Out.Stat.RecipeList[kk+1]), ADR(gRecipe_Ctrl.Out.Stat.RecipeList[kk]));
				strcpy(ADR(gRecipe_Ctrl.Out.Stat.RecipeList[kk]), ADR(SaveFileName));
			END_IF
			kk := kk+1;
			IF (Changed) THEN
				Changed	:= FALSE;
				kk 		:= 0;
			END_IF
			UNTIL (kk = (gRecipe_Ctrl.In.Stat.FileHandling.DirectoryInformation.NrFiles - 1))
		END_REPEAT
	END_IF

END_ACTION

(*Check error actions*)
ACTION Action_CheckError:

	//Check if there are error from low level tasks
	IF (MainState <> C_MS_RECIPE_HAND_ACK_ERROR) THEN
		IF (gRecipe_Ctrl.In.Stat.FileHandling.Error.Number <> 0) THEN
			//Copy eeror information
			gRecipe_Ctrl.Out.Stat.Error	:= gRecipe_Ctrl.In.Stat.FileHandling.Error;
			//Go to error state
			MainState					:= C_MS_RECIPE_HAND_ERROR;
		END_IF
		IF (gRecipe_Ctrl.In.Stat.CsvHandling.Error.Number <> 0) THEN
			//Copy eeror information
			gRecipe_Ctrl.Out.Stat.Error	:= gRecipe_Ctrl.In.Stat.CsvHandling.Error;
			//Go to error state
			MainState					:= C_MS_RECIPE_HAND_ERROR;
		END_IF
	END_IF

END_ACTION
```

### Package Logical/CuttingTable/RecipeHandling/CsvHandling - CSV handling program
